# B&R Automation Studio project mappFramework (part 10)

#### Set_SetupTeardown.c - not listed in the package file held
```c
#include <bur/plctypes.h>

#ifdef _DEFAULT_INCLUDES
#include <AsDefault.h>
#endif

#include "UnitTest.h"
#include <stdbool.h>
#include <string.h>

_SETUP_SET(void)
{
	/* TODO:  add code running before test set here */
	TEST_DONE;
}

_TEARDOWN_SET(void)
{
	/* TODO:  add code running after test set here */
	TEST_DONE;
}

_SETUP_TEST(void)
{
    TestState = 0;
    FileNumber = 0;

    HmiFile_UT.Parameters.Fifo.Enable = false;
    HmiFile_UT.Parameters.Fifo.ScanInterval = 60;
    strcpy(HmiFile_UT.Parameters.Fifo.DeviceName, "mappUserXFiles");

    switch (SetupState)
    {
        case 0:
            DirInfo_UT.enable = true;
            DirInfo_UT.pDevice = (UDINT)&"mappUserXFiles";
            DirInfo_UT.pPath = (UDINT)&"";
            DirInfo(&DirInfo_UT);
            TEST_BUSY_CONDITION(DirInfo_UT.status == 65535);
            TEST_ABORT_CONDITION(DirInfo_UT.status != 0);
            NumberOfFiles = DirInfo_UT.filenum;
            CurrentFile = 0;
            SetupState = (NumberOfFiles == 0) ? 100 : 1;
            break;

        case 1:
            DirRead_UT.enable = true;
            DirRead_UT.pDevice = DirInfo_UT.pDevice;
            DirRead_UT.entry = 0;
            DirRead_UT.option = fiFILE;
            DirRead_UT.pData = (UDINT)&fileInfo;
            DirRead_UT.data_len = sizeof(fileInfo);
            DirRead(&DirRead_UT);
            TEST_BUSY_CONDITION(DirRead_UT.status == 65535);
            TEST_ABORT_CONDITION(DirRead_UT.status != 0);
            SetupState = 2;
            break;

        case 2:
            FileDelete_UT.enable = true;
            FileDelete_UT.pDevice = DirInfo_UT.pDevice;
            FileDelete_UT.pName = (UDINT)&fileInfo.Filename;
            FileDelete(&FileDelete_UT);
            TEST_BUSY_CONDITION(FileDelete_UT.status == 65535);
            TEST_ABORT_CONDITION(FileDelete_UT.status != 0);

            CurrentFile++;
            SetupState = (CurrentFile >= NumberOfFiles) ? 100 : 1;
            break;

        case 100:
            TEST_DONE;
    }
    TEST_BUSY;
}

_TEARDOWN_TEST(void)
{
    HmiFile_UT.Parameters.Fifo.Enable = false;
    HmiFile_UT.Parameters.Fifo.ScanInterval = 60;
    TestState = 0;
    SetupState = 0;
	TEST_DONE;
}

_TEST FIFO_20(void)
{
    switch (TestState)
    {
        // Arrange
        case 0:
            FileCreate_UT.enable = true;
            FileCreate_UT.pDevice = (UDINT)&"mappUserXFiles";
            snprintf2(FileName, sizeof(FileName), "TestFile%d.txt", FileNumber);
            FileCreate_UT.pFile = (UDINT)&FileName;
            FileCreate(&FileCreate_UT);

            TEST_BUSY_CONDITION(FileCreate_UT.status == 65535);
            TEST_ABORT_CONDITION(FileCreate_UT.status != 0);
            TestState = 1;
            break;

        case 1:
            FileClose_UT.enable = true;
            FileClose_UT.ident = FileCreate_UT.ident;
            FileClose(&FileClose_UT);

            TEST_BUSY_CONDITION(FileClose_UT.status == 65535);
            TEST_ABORT_CONDITION(FileClose_UT.status != 0);

            FileNumber++;
            TestState = (FileNumber >= 20) ? 10 : 0;
            break;

        // Act
        case 10:
            HmiFile_UT.Parameters.Fifo.Enable = true;
            strcpy(HmiFile_UT.Parameters.Fifo.DeviceName, "mappUserXFiles");
            HmiFile_UT.Parameters.Fifo.FifoType = FILE_FIFO_NUM_OF_FILES;
            HmiFile_UT.Parameters.Fifo.MaxNumberOfFiles = 10;
            HmiFile_UT.Parameters.Fifo.ScanInterval = 0;
            TEST_BUSY_CONDITION(HmiFile_UT.Status.DeleteStep == FILE_DELETE_WAIT);
            TestState = 100;
            break;

        // Assert
        case 100:
            TEST_BUSY_CONDITION(HmiFile_UT.Status.DeleteStep != FILE_DELETE_WAIT);
            HmiFile_UT.Parameters.Fifo.Enable = false;

            DirInfo_UT.enable = true;
            DirInfo_UT.pDevice = (UDINT)&"mappUserXFiles";
            DirInfo_UT.pPath = (UDINT)&"";
            DirInfo(&DirInfo_UT);
            TEST_BUSY_CONDITION(DirInfo_UT.status == 65535);
            TEST_ABORT_CONDITION(DirInfo_UT.status != 0);
            TEST_ASSERT_EQUAL_INT(HmiFile_UT.Parameters.Fifo.MaxNumberOfFiles, DirInfo_UT.filenum);
            TEST_DONE;
            break;
    }
    TEST_BUSY;
}

_TEST FIFO_60(void)
{
    switch (TestState)
    {
        // Arrange
        case 0:
            FileCreate_UT.enable = true;
            FileCreate_UT.pDevice = (UDINT)&"mappUserXFiles";
            snprintf2(FileName, sizeof(FileName), "TestFile%d.txt", FileNumber);
            FileCreate_UT.pFile = (UDINT)&FileName;
            FileCreate(&FileCreate_UT);

            TEST_BUSY_CONDITION(FileCreate_UT.status == 65535);
            TEST_ABORT_CONDITION(FileCreate_UT.status != 0);
            TestState = 1;
            break;

        case 1:
            FileClose_UT.enable = true;
            FileClose_UT.ident = FileCreate_UT.ident;
            FileClose(&FileClose_UT);

            TEST_BUSY_CONDITION(FileClose_UT.status == 65535);
            TEST_ABORT_CONDITION(FileClose_UT.status != 0);

            FileNumber++;
            TestState = (FileNumber >= 60) ? 10 : 0;
            break;

        // Act
        case 10:
            HmiFile_UT.Parameters.Fifo.Enable = true;
            strcpy(HmiFile_UT.Parameters.Fifo.DeviceName, "mappUserXFiles");
            HmiFile_UT.Parameters.Fifo.FifoType = FILE_FIFO_NUM_OF_FILES;
            HmiFile_UT.Parameters.Fifo.MaxNumberOfFiles = 15;
            HmiFile_UT.Parameters.Fifo.ScanInterval = 0;
            TEST_BUSY_CONDITION(HmiFile_UT.Status.DeleteStep == FILE_DELETE_WAIT);
            TestState = 100;
            break;

        // Assert
        case 100:
            TEST_BUSY_CONDITION(HmiFile_UT.Status.DeleteStep != FILE_DELETE_WAIT);
            HmiFile_UT.Parameters.Fifo.Enable = false;

            DirInfo_UT.enable = true;
            DirInfo_UT.pDevice = (UDINT)&"mappUserXFiles";
            DirInfo_UT.pPath = (UDINT)&"";
            DirInfo(&DirInfo_UT);
            TEST_BUSY_CONDITION(DirInfo_UT.status == 65535);
            TEST_ABORT_CONDITION(DirInfo_UT.status != 0);
            TEST_ASSERT_EQUAL_INT(HmiFile_UT.Parameters.Fifo.MaxNumberOfFiles, DirInfo_UT.filenum);
            TEST_DONE;
            break;

    }
    TEST_BUSY;
}

_TEST FIFO_140(void)
{
    switch (TestState)
    {
        // Arrange
        case 0:
            FileCreate_UT.enable = true;
            FileCreate_UT.pDevice = (UDINT)&"mappUserXFiles";
            snprintf2(FileName, sizeof(FileName), "TestFile%d.txt", FileNumber);
            FileCreate_UT.pFile = (UDINT)&FileName;
            FileCreate(&FileCreate_UT);

            TEST_BUSY_CONDITION(FileCreate_UT.status == 65535);
            TEST_ABORT_CONDITION(FileCreate_UT.status != 0);
            TestState = 1;
            break;

        case 1:
            FileClose_UT.enable = true;
            FileClose_UT.ident = FileCreate_UT.ident;
            FileClose(&FileClose_UT);

            TEST_BUSY_CONDITION(FileClose_UT.status == 65535);
            TEST_ABORT_CONDITION(FileClose_UT.status != 0);

            FileNumber++;
            TestState = (FileNumber >= 140) ? 10 : 0;
            break;

        // Act
        case 10:
            HmiFile_UT.Parameters.Fifo.Enable = true;
            strcpy(HmiFile_UT.Parameters.Fifo.DeviceName, "mappUserXFiles");
            HmiFile_UT.Parameters.Fifo.FifoType = FILE_FIFO_NUM_OF_FILES;
            HmiFile_UT.Parameters.Fifo.MaxNumberOfFiles = 15;
            HmiFile_UT.Parameters.Fifo.ScanInterval = 0;
            TEST_BUSY_CONDITION(HmiFile_UT.Status.DeleteStep == FILE_DELETE_WAIT);
            TestState = 100;
            break;

        // Assert
        case 100:
            TEST_BUSY_CONDITION(HmiFile_UT.Status.DeleteStep != FILE_DELETE_WAIT);
            HmiFile_UT.Parameters.Fifo.Enable = false;

            DirInfo_UT.enable = true;
            DirInfo_UT.pDevice = (UDINT)&"mappUserXFiles";
            DirInfo_UT.pPath = (UDINT)&"";
            DirInfo(&DirInfo_UT);
            TEST_BUSY_CONDITION(DirInfo_UT.status == 65535);
            TEST_ABORT_CONDITION(DirInfo_UT.status != 0);
            TEST_ASSERT_EQUAL_INT(HmiFile_UT.Parameters.Fifo.MaxNumberOfFiles, DirInfo_UT.filenum);
            TEST_DONE;
            break;

    }
    TEST_BUSY;
}

_TEST FIFO_MaxFiles60(void)
{
    switch (TestState)
    {
        // Arrange
        case 0:
            FileCreate_UT.enable = true;
            FileCreate_UT.pDevice = (UDINT)&"mappUserXFiles";
            snprintf2(FileName, sizeof(FileName), "TestFile%d.txt", FileNumber);
            FileCreate_UT.pFile = (UDINT)&FileName;
            FileCreate(&FileCreate_UT);

            TEST_BUSY_CONDITION(FileCreate_UT.status == 65535);
            TEST_ABORT_CONDITION(FileCreate_UT.status != 0);
            TestState = 1;
            break;

        case 1:
            FileClose_UT.enable = true;
            FileClose_UT.ident = FileCreate_UT.ident;
            FileClose(&FileClose_UT);

            TEST_BUSY_CONDITION(FileClose_UT.status == 65535);
            TEST_ABORT_CONDITION(FileClose_UT.status != 0);

            FileNumber++;
            TestState = (FileNumber >= 100) ? 10 : 0;
            break;

        // Act
        case 10:
            HmiFile_UT.Parameters.Fifo.Enable = true;
            strcpy(HmiFile_UT.Parameters.Fifo.DeviceName, "mappUserXFiles");
            HmiFile_UT.Parameters.Fifo.FifoType = FILE_FIFO_NUM_OF_FILES;
            HmiFile_UT.Parameters.Fifo.MaxNumberOfFiles = 60;
            HmiFile_UT.Parameters.Fifo.ScanInterval = 0;
            TEST_BUSY_CONDITION(HmiFile_UT.Status.DeleteStep == FILE_DELETE_WAIT);
            TestState = 100;
            break;

        // Assert
        case 100:
            TEST_BUSY_CONDITION(HmiFile_UT.Status.DeleteStep != FILE_DELETE_WAIT);
            HmiFile_UT.Parameters.Fifo.Enable = false;

            DirInfo_UT.enable = true;
            DirInfo_UT.pDevice = (UDINT)&"mappUserXFiles";
            DirInfo_UT.pPath = (UDINT)&"";
            DirInfo(&DirInfo_UT);
            TEST_BUSY_CONDITION(DirInfo_UT.status == 65535);
            TEST_ABORT_CONDITION(DirInfo_UT.status != 0);
            TEST_ASSERT_EQUAL_INT(HmiFile_UT.Parameters.Fifo.MaxNumberOfFiles, DirInfo_UT.filenum);
            TEST_DONE;
            break;

    }
    TEST_BUSY;
}

_TEST FIFO_MaxFiles120(void)
{
    switch (TestState)
    {
        // Arrange
        case 0:
            FileCreate_UT.enable = true;
            FileCreate_UT.pDevice = (UDINT)&"mappUserXFiles";
            snprintf2(FileName, sizeof(FileName), "TestFile%d.txt", FileNumber);
            FileCreate_UT.pFile = (UDINT)&FileName;
            FileCreate(&FileCreate_UT);

            TEST_BUSY_CONDITION(FileCreate_UT.status == 65535);
            TEST_ABORT_CONDITION(FileCreate_UT.status != 0);
            TestState = 1;
            break;

        case 1:
            FileClose_UT.enable = true;
            FileClose_UT.ident = FileCreate_UT.ident;
            FileClose(&FileClose_UT);

            TEST_BUSY_CONDITION(FileClose_UT.status == 65535);
            TEST_ABORT_CONDITION(FileClose_UT.status != 0);

            FileNumber++;
            TestState = (FileNumber >= 200) ? 10 : 0;
            break;

        // Act
        case 10:
            HmiFile_UT.Parameters.Fifo.Enable = true;
            strcpy(HmiFile_UT.Parameters.Fifo.DeviceName, "mappUserXFiles");
            HmiFile_UT.Parameters.Fifo.FifoType = FILE_FIFO_NUM_OF_FILES;
            HmiFile_UT.Parameters.Fifo.MaxNumberOfFiles = 120;
            HmiFile_UT.Parameters.Fifo.ScanInterval = 0;
            TEST_BUSY_CONDITION(HmiFile_UT.Status.DeleteStep == FILE_DELETE_WAIT);
            TestState = 100;
            break;

        // Assert
        case 100:
            TEST_BUSY_CONDITION(HmiFile_UT.Status.DeleteStep != FILE_DELETE_WAIT);
            HmiFile_UT.Parameters.Fifo.Enable = false;

            DirInfo_UT.enable = true;
            DirInfo_UT.pDevice = (UDINT)&"mappUserXFiles";
            DirInfo_UT.pPath = (UDINT)&"";
            DirInfo(&DirInfo_UT);
            TEST_BUSY_CONDITION(DirInfo_UT.status == 65535);
            TEST_ABORT_CONDITION(DirInfo_UT.status != 0);
            TEST_ASSERT_EQUAL_INT(HmiFile_UT.Parameters.Fifo.MaxNumberOfFiles, DirInfo_UT.filenum);
            TEST_DONE;
            break;

    }
    TEST_BUSY;
}

_TEST FIFO_MaxFolderSize_60Files(void)
{
    switch (TestState)
    {
        // Arrange
        case 0:
            FileCreate_UT.enable = true;
            FileCreate_UT.pDevice = (UDINT)&"mappUserXFiles";
            snprintf2(FileName, sizeof(FileName), "TestFile%d.txt", FileNumber);
            FileCreate_UT.pFile = (UDINT)&FileName;
            FileCreate(&FileCreate_UT);

            TEST_BUSY_CONDITION(FileCreate_UT.status == 65535);
            TEST_ABORT_CONDITION(FileCreate_UT.status != 0);
            TestState = 1;
            break;

        case 1:
            FileWrite_UT.enable = true;
            FileWrite_UT.ident = FileCreate_UT.ident;
            FileWrite_UT.offset = 0;
            FileWrite_UT.pSrc = &testData;
            FileWrite_UT.len = sizeof(testData);
            FileWrite(&FileWrite_UT);
            TEST_BUSY_CONDITION(FileWrite_UT.status == 65535);
            TEST_ABORT_CONDITION(FileWrite_UT.status != 0);
            TestState = 2;
            break;

        case 2:
            FileClose_UT.enable = true;
            FileClose_UT.ident = FileCreate_UT.ident;
            FileClose(&FileClose_UT);

            TEST_BUSY_CONDITION(FileClose_UT.status == 65535);
            TEST_ABORT_CONDITION(FileClose_UT.status != 0);

            FileNumber++;
            TestState = (FileNumber >= 60) ? 10 : 0;
            break;

        // Act
        case 10:
            HmiFile_UT.Parameters.Fifo.Enable = true;
            strcpy(HmiFile_UT.Parameters.Fifo.DeviceName, "mappUserXFiles");
            HmiFile_UT.Parameters.Fifo.FifoType = FILE_FIFO_SIZE_OF_FOLDER;
            HmiFile_UT.Parameters.Fifo.MaxFolderSize = 5 * 1024;
            HmiFile_UT.Parameters.Fifo.ScanInterval = 0;
            TEST_BUSY_CONDITION(HmiFile_UT.Status.DeleteStep == FILE_DELETE_WAIT);
            TestState = 100;
            break;

        // Assert
        case 100:
            TEST_BUSY_CONDITION(HmiFile_UT.Status.DeleteStep != FILE_DELETE_WAIT);
            HmiFile_UT.Parameters.Fifo.Enable = false;

            DirInfo_UT.enable = true;
            DirInfo_UT.pDevice = (UDINT)&"mappUserXFiles";
            DirInfo_UT.pPath = (UDINT)&"";
            DirInfo(&DirInfo_UT);
            TEST_BUSY_CONDITION(DirInfo_UT.status == 65535);
            TEST_ABORT_CONDITION(DirInfo_UT.status != 0);
            TEST_ASSERT_EQUAL_INT(5, DirInfo_UT.filenum);
            TEST_DONE;
            break;

    }
    TEST_BUSY;
}

/*
B+R UnitTest: This is generated code.
Do not edit! Do not move!
Description: UnitTest Testprogramm infrastructure (TestSet).
LastUpdated: 2022-04-25 15:09:32Z
By B+R UnitTest Helper Version: 2.0.1.59
*/
UNITTEST_FIXTURES(fixtures)
{
    new_TestFixture("FIFO_20", FIFO_20),
    new_TestFixture("FIFO_60", FIFO_60),
    new_TestFixture("FIFO_140", FIFO_140),
    new_TestFixture("FIFO_MaxFiles60", FIFO_MaxFiles60),
    new_TestFixture("FIFO_MaxFiles120", FIFO_MaxFiles120),
    new_TestFixture("FIFO_MaxFolderSize_60Files", FIFO_MaxFolderSize_60Files),

};

UNITTEST_CALLER_COMPLETE_EXPLICIT(Set_SetupTeardown, "Set_SetupTeardown", setupTest, teardownTest, fixtures, setupSet, teardownSet, 0);
```

### Package Logical/UnitTest/Recipe - Package for mapp Recipe Framework

### Program Logical/UnitTest/Recipe/RecipeMgrUnitTest (ANSIC) - Unit Tests for FileMgr

- RecipeMgr.typ (reference to Logical/Infrastructure/Recipe/RecipeMgr/RecipeMgr.typ)

- RecipeMgr.var (reference to Logical/Infrastructure/Recipe/RecipeMgr/RecipeMgr.var)

- CommonVariables.var (reference to Logical/UnitTest/Common/CommonUT/CommonVariables.var)

- Set_Common.c (reference to Logical/UnitTest/Common/CommonUT/Set_Common.c)

#### variables.var - Name the suite and add PVs for the program
```iecst
(********************************************************************
 * COPYRIGHT --
 ********************************************************************
 * Program: utTemplate_automated
 * File: variables.var
 * Author: -
 * Created: -
 ********************************************************************
 * Local variables of program utTemplate_automated
 ********************************************************************)
(*Describe the test*)
VAR
	Testsuite : UtMgrTestSuite := (Name:='RecipeMgr',Description:='RecipeMgr Unit Tests',MetaInformation:='Meta');
END_VAR
(*Variables used in the tests*)
VAR
	cycleCount : {REDUND_UNREPLICABLE} USINT;
	pMachineSettings : REFERENCE TO MachineSettingsType;
	MachineSettingsSize : {REDUND_UNREPLICABLE} UDINT;
	pParameters : REFERENCE TO ParametersType;
	ParameterSize : {REDUND_UNREPLICABLE} UDINT;
	LastSelectedIndex : UDINT;
	SetupState : USINT;
	FileName : STRING[24];
	NumberOfFiles : UINT;
	CurrentFile : UINT;
	fileInfo : fiDIR_READ_DATA;
	DirInfo_UT : DirInfo;
	DirRead_UT : DirRead;
	FileDelete_UT : FileDelete;
	FileCopy_UT : FileCopy;
END_VAR
```

#### testSuite.h
```c
#ifndef __TEST_SUITE_H__
#define __TEST_SUITE_H__

bool RecipeExists(char* recipeName);
bool SelectRecipe(char* wantedRecipe);
testStatusEnum RemoveNonDefaultFiles(char* filter, char* selectFile, const USINT categoryIndex, const char* category);

#endif
```

#### testSuite.c
```c
/********************************************************************
 * COPYRIGHT --
 ********************************************************************
 * Program: -
 * Author:
 * Created:
 ********************************************************************
 * Test registration and handshake
 ********************************************************************/

#include <bur/plctypes.h>

#ifdef _DEFAULT_INCLUDES
#include <AsDefault.h>
#endif

#include "UnitTest.h"
#include <string.h>
#include <stdbool.h>

void _INIT initTestSuite(void)
{
	Testsuite.Enable = 1;
	utInit(&Testsuite);

	CommonTestsuite.Enable = 1;
	utInit(&CommonTestsuite);

	strcpy((char*)&FileDeviceName, "mappRecipeFiles");
	strcpy((char*)&TextNameSpace, "mappFramework/Recipe/Alarms");
	strcpy((char*)&TextID, "SaveFailed");
	strcpy((char*)&HmiRecipe.Parameters.DeviceName, "mappRecipeFiles");

	PV_xgetadr("RecipeMgr:MachineSettings", (void*)&pMachineSettings, &MachineSettingsSize);
	PV_xgetadr("RecipeMgr:Parameters", (void*)&pParameters, &ParameterSize);

	LastSelectedIndex++;
}

void _CYCLIC cyclicWithTest(void)
{
	utCyclic(&Testsuite);
	if (Testsuite.Informational.LastKnownPassedLocation.TestCaseName != 0)
		strcpy((char*)&LastTestCase, (char*)Testsuite.Informational.LastKnownPassedLocation.TestCaseName);
	if (Testsuite.Informational.LastKnownPassedLocation.TestSetName != 0)
		strcpy((char*)&LastTestSet, (char*)Testsuite.Informational.LastKnownPassedLocation.TestSetName);
	if (Testsuite.Informational.LastKnownPassedLocation.File != 0)
		strcpy((char*)&LastTestFile, (char*)Testsuite.Informational.LastKnownPassedLocation.File);
}

void _EXIT exitTestSuite(void)
{
	utExit(&Testsuite);
}

bool RecipeExists(char* recipeName)
{
	for (USINT i = 0; i<(sizeof(MpRecipeUIConnect.Recipe.List.Names)/sizeof(MpRecipeUIConnect.Recipe.List.Names[0])); i++)
	{
		if (strcmp(recipeName, MpRecipeUIConnect.Recipe.List.Names[i]) == 0)
		{
			return true;
		}
	}
	return false;
}

bool SelectRecipe(char* wantedRecipe)
{
	if (((MpRecipeUIConnect.Status != mpRECIPE_UI_STATUS_IDLE) && (MpRecipeUIConnect.Status != mpRECIPE_UI_STATUS_ERROR)) &&
		(strcmp(wantedRecipe, HmiRecipe.Status.SelectedRecipe) != 0)) return false;

	for (USINT i=0; i <= MpRecipeUIConnect.Recipe.List.MaxSelection; i++)
	{
		if (strcmp(wantedRecipe, MpRecipeUIConnect.Recipe.List.Names[i]) == 0)
			MpRecipeUIConnect.Recipe.List.SelectedIndex = i;
	}

	return (strcmp(wantedRecipe, HmiRecipe.Status.SelectedRecipe) == 0);
}

testStatusEnum RemoveNonDefaultFiles(char* filter, char* selectFile, const char* category)
{
	switch (SetupState)
	{
		case 0:
			DirInfo_UT.enable = true;
			DirInfo_UT.pDevice = (UDINT)&"mappRecipeFiles";
			DirInfo_UT.pPath = (UDINT)&"";
			DirInfo(&DirInfo_UT);
			TEST_BUSY_CONDITION(DirInfo_UT.status == 65535);
			TEST_ABORT_CONDITION(DirInfo_UT.status != 0);
			NumberOfFiles = DirInfo_UT.filenum;
			CurrentFile = 0;
			SetupState = (NumberOfFiles == 0) ? 100 : 1;
			break;

		case 1:
			DirRead_UT.enable = true;
			DirRead_UT.pDevice = DirInfo_UT.pDevice;
			DirRead_UT.entry = CurrentFile;
			DirRead_UT.option = fiFILE;
			DirRead_UT.pData = (UDINT)&fileInfo;
			DirRead_UT.data_len = sizeof(fileInfo);
			DirRead(&DirRead_UT);
			TEST_BUSY_CONDITION(DirRead_UT.status == 65535);
			TEST_ABORT_CONDITION(DirRead_UT.status != 0);
			SetupState = 2;
			break;

		case 2:
			if ((strcmp("Default.par", (char*)fileInfo.Filename) == 0) ||
				(strcmp("Machine.mcfg", (char*)fileInfo.Filename) == 0))
			{
				CurrentFile++;
				SetupState = (CurrentFile >= NumberOfFiles) ? 10 : 1;
				break;
			}
			FileDelete_UT.enable = true;
			FileDelete_UT.pDevice = DirInfo_UT.pDevice;
			FileDelete_UT.pName = (UDINT)&fileInfo.Filename;
			FileDelete(&FileDelete_UT);
			TEST_BUSY_CONDITION(FileDelete_UT.status == 65535);
			TEST_ABORT_CONDITION(FileDelete_UT.status != 0);

			NumberOfFiles--;
			SetupState = (CurrentFile >= NumberOfFiles) ? 10 : 1;
			break;

		case 10:
			strcpy((char*)&HmiRecipe.Parameters.DeviceName, "mappRecipeFiles");
			strcpy((char*)&MpRecipeUIConnect.Recipe.Filter, filter);
			MpRecipeUIConnect.Recipe.Refresh = true;
			strcpy((char*)&HmiRecipe.Parameters.Category, category);
			TEST_BUSY_CONDITION(MpRecipeUIConnect.Status != mpRECIPE_UI_STATUS_REFRESH)
			MpRecipeUIConnect.Recipe.Refresh = false;
			SetupState = 11;
			break;

		case 11:
			TEST_BUSY_CONDITION(MpRecipeUIConnect.Status != mpRECIPE_UI_STATUS_IDLE)
			TEST_BUSY_CONDITION(!RecipeExists(selectFile));
			TEST_BUSY_CONDITION(HmiRecipe.Status.HMIcommand != REC_HMI_WAIT)
			TEST_ABORT_CONDITION(pParameters == NULL);
			SetupState = 100;
			break;

		case 100:
			cycleCount = 0;
			TestState = TEST_ARRANGE;
			SetupState = 0;
			TEST_DONE;
	}
	TEST_BUSY;
}
```

#### autoGeneratedFile.c - Auto generated code - list of all test sets in the program
```c
/*
B+R UnitTest: This is generated code.
Do not edit! Do not move!
Description: UnitTest Testprogramm infrastructure (List of TestSets).
LastUpdated: 2022-11-02 11:34:44Z
By B+R UnitTest Helper Version: 2.0.1.59
*/
#include "UnitTest.h"

UNITTEST_TESTSET_DECLARATION  Set_Common;
UNITTEST_TESTSET_DECLARATION  Set_RecipeParameters;
UNITTEST_TESTSET_DECLARATION  Set_RecipeMachineSettings;

UNITTEST_TESTSET_FIXTURES(utTestSets)
{
	new_TestSet(Set_Common),
	new_TestSet(Set_RecipeParameters),
	new_TestSet(Set_RecipeMachineSettings),
};
UNTITTEST_TESTSET_HANDLER();
```

#### Set_RecipeParameters.c
```c
#include <bur/plctypes.h>

#ifdef _DEFAULT_INCLUDES
#include <AsDefault.h>
#endif

#include "UnitTest.h"
#include <stdbool.h>
#include <string.h>
#include <stdlib.h>
#include "testSuite.h"

#define TIMEOUT_TEST_CASE                                   \
    if (cycleCount >= 254)                                  \
    {                                                       \
        char abortMessage[80];                              \
        char substate[10];                                  \
        memset(abortMessage, 0, sizeof(abortMessage));      \
        memset(substate, 0, sizeof(substate));              \
        itoa(ActSubState, substate, 10);                    \
        strcpy(abortMessage, "Timeout in ActSubState = ");  \
        strcat(abortMessage, substate);                     \
        TEST_FAIL(abortMessage);                            \
        TEST_DONE;                                          \
    }

_SETUP_SET(void)
{
    return RemoveNonDefaultFiles("*.par", "Default.par", PARAMETERS_CATEGORY);
}

_TEARDOWN_SET(void)
{
    SetupState = 0;
    TEST_DONE;
}

_SETUP_TEST(void)
{
    ArrangeSubState = 0;
    ActSubState = 0;
    AssertSubState = 0;
    return RemoveNonDefaultFiles("*.par", "Default.par", PARAMETERS_CATEGORY);
}

_TEARDOWN_TEST(void)
{
    memset(&HmiRecipe.Commands, 0, sizeof(HmiRecipe.Commands));
    MpRecipeUIConnect.Recipe.Load = false;
    TEST_BUSY_CONDITION(!SelectRecipe("Default.par"));

    if (MpRecipeUIConnect.Status == mpRECIPE_UI_STATUS_ERROR)
    {
        MpRecipeUIConnect.Recipe.Refresh = true;
    }
    TEST_BUSY_CONDITION(MpRecipeUIConnect.Status != mpRECIPE_UI_STATUS_IDLE)
    MpRecipeUIConnect.Recipe.Refresh = false;

    TEST_DONE;
}

_CYCLIC_SET(void)
{
    cycleCount++;
}

_TEST DefaultValues(void)
{
    TIMEOUT_TEST_CASE
    switch (TestState)
    {
        case TEST_ARRANGE:
            // set MachineSettings through the pointer
            memset(pParameters, 0, sizeof(*pParameters));
            TEST_BUSY_CONDITION(!SelectRecipe("Default.par"));
            TEST_BUSY_CONDITION(MpRecipeUIConnect.Status != mpRECIPE_UI_STATUS_IDLE);
            TEST_BUSY_CONDITION(HmiRecipe.Status.HMIcommand != REC_HMI_WAIT);
            TestState = TEST_ACT;
            break;

        case TEST_ACT:
            switch (ActSubState)
            {
                case 0:
                    MpRecipeUIConnect.Recipe.Load = true;
                    TEST_BUSY_CONDITION(MpRecipeUIConnect.Status != mpRECIPE_UI_STATUS_LOAD);
                    MpRecipeUIConnect.Recipe.Load = false;
                    ActSubState = 1;
                    break;

                case 1:
                    TEST_BUSY_CONDITION(MpRecipeUIConnect.Status != mpRECIPE_UI_STATUS_IDLE);
                    HmiRecipe.Commands.LoadRecipe = true;
                    TEST_BUSY_CONDITION(HmiRecipe.Status.ProductRecipeLoaded == true);
                    TEST_BUSY_CONDITION(HmiRecipe.Status.HMIcommand == REC_HMI_WAIT);
                    HmiRecipe.Commands.LoadRecipe = false;
                    ActSubState = 2;
                    break;

                case 2:
                    TEST_BUSY_CONDITION(HmiRecipe.Status.ProductRecipeLoaded == false);
                    TEST_BUSY_CONDITION(HmiRecipe.Status.HMIcommand != REC_HMI_WAIT);
                    TestState = TEST_ASSERT;
                    break;
            }
            break;

        case TEST_ASSERT:
            TEST_ASSERT(Parameters.AddParametersHere1);
            TEST_ASSERT_EQUAL_STRING("two", Parameters.AddParametersHere2);
            TEST_ASSERT_DOUBLE_WITHIN(0.0001, 3.3, Parameters.AddParametersHere3);
            TEST_ASSERT_DOUBLE_WITHIN(0.0001, 4.4, Parameters.AddParametersHere4);
            TEST_ASSERT_DOUBLE_WITHIN(0.0001, 5.5, Parameters.AddParametersHere5);
            TEST_DONE;
            break;
    }
    TEST_BUSY;
}

_TEST CreateNew(void)
{
    TIMEOUT_TEST_CASE
    switch (TestState)
    {
        case TEST_ARRANGE:
            strcpy(HmiRecipe.Parameters.FileName, "test");
            TEST_BUSY_CONDITION(MpRecipeUIConnect.Status != mpRECIPE_UI_STATUS_IDLE);
            TEST_BUSY_CONDITION(HmiRecipe.Status.HMIcommand != REC_HMI_WAIT);
            TestState = TEST_ACT;
            break;

        case TEST_ACT:
            if (MpRecipeUIConnect.Status == mpRECIPE_UI_STATUS_ERROR)
            {
                TEST_FAIL("MpRecipeUIConnect in error state");
            }
            switch (ActSubState)
            {
                case 0:
                    HmiRecipe.Commands.CreateRecipe = true;
                    TEST_BUSY_CONDITION(MpRecipeUIConnect.Status != mpRECIPE_UI_STATUS_CREATE);
                    HmiRecipe.Commands.CreateRecipe = false;
                    ActSubState = 1;
                    break;

                case 1:
                    TEST_BUSY_CONDITION(MpRecipeUIConnect.Status != mpRECIPE_UI_STATUS_IDLE);
                    TEST_BUSY_CONDITION(HmiRecipe.Status.ProductRecipeLoaded == false);
                    ActSubState = 2;
                    break;

                case 2:
                    TEST_BUSY_CONDITION(MpRecipeUIConnect.Status == mpRECIPE_UI_STATUS_REFRESH);
                    ActSubState = 3;
                    break;

                case 3:
                    TEST_BUSY_CONDITION(MpRecipeUIConnect.Status != mpRECIPE_UI_STATUS_IDLE);
                    TestState = TEST_ASSERT;
                    break;
            }
            break;

        case TEST_ASSERT:
            TEST_ASSERT(RecipeExists("test.par"));
            TEST_DONE;
            break;
    }

    TEST_BUSY;
}

_TEST CreateExisting(void)
{
    TIMEOUT_TEST_CASE
    switch (TestState)
    {
        case TEST_ARRANGE:
            strcpy(HmiRecipe.Parameters.FileName, "Default");
            TEST_BUSY_CONDITION(MpRecipeUIConnect.Status != mpRECIPE_UI_STATUS_IDLE);
            TEST_BUSY_CONDITION(HmiRecipe.Status.HMIcommand != REC_HMI_WAIT);
            TestState = TEST_ACT;
            break;

        case TEST_ACT:
            TestState = TEST_ASSERT;
            break;

        case TEST_ASSERT:
            HmiRecipe.Commands.CreateRecipe = false;
            TEST_ASSERT(HmiRecipe.Status.FileDuplicate);
            TEST_ASSERT(RecipeExists("Default.par"));
            TEST_DONE;
            break;
    }

    TEST_BUSY;
}

_TEST CreateNonExisting(void)
{
    TIMEOUT_TEST_CASE

    switch (TestState)
    {
        case TEST_ARRANGE:
            strcpy(HmiRecipe.Parameters.FileName, "test2");
            TEST_BUSY_CONDITION(MpRecipeUIConnect.Status != mpRECIPE_UI_STATUS_IDLE);
            TEST_BUSY_CONDITION(HmiRecipe.Status.HMIcommand != REC_HMI_WAIT);
            TestState = TEST_ACT;
            break;

        case TEST_ACT:
            TestState = TEST_ASSERT;
            break;

        case TEST_ASSERT:
            HmiRecipe.Commands.CreateRecipe = false;
            TEST_ASSERT(!HmiRecipe.Status.FileDuplicate);
            TEST_ASSERT(!RecipeExists("test2.par"));
            TEST_DONE;
            break;
    }
    TEST_BUSY;
}

_TEST CreateActive(void)
{
    TIMEOUT_TEST_CASE
    switch (TestState)
    {
        case TEST_ARRANGE:
            strcpy(HmiRecipe.Parameters.FileName, strtok(HmiRecipe.Status.LastLoadedProductRecipe, "."));
            TEST_BUSY_CONDITION(MpRecipeUIConnect.Status != mpRECIPE_UI_STATUS_IDLE);
            TEST_BUSY_CONDITION(HmiRecipe.Status.HMIcommand != REC_HMI_WAIT);
            TestState = TEST_ACT;
            break;

        case TEST_ACT:
            TestState = TEST_ASSERT;
            break;

        case TEST_ASSERT:
            HmiRecipe.Commands.CreateRecipe = false;
            TEST_ASSERT(HmiRecipe.Status.FileDuplicate);
            TEST_ASSERT(RecipeExists(HmiRecipe.Status.LastLoadedProductRecipe));
            TEST_DONE;
            break;
    }
    TEST_BUSY;
}

_TEST PreviewShouldNotAffectActive(void)
{
    TIMEOUT_TEST_CASE
    switch (TestState)
    {
        case TEST_ARRANGE:
            ParametersEdit.AddParametersHere1 = false;
            strcpy(ParametersEdit.AddParametersHere2, "testing preview");
            ParametersEdit.AddParametersHere3 = 12.56;
            ParametersEdit.AddParametersHere4 = 134.876;
            ParametersEdit.AddParametersHere5 = 87.4567;
            strcpy(HmiRecipe.Parameters.FileName, "preview");
            TEST_BUSY_CONDITION(MpRecipeUIConnect.Status != mpRECIPE_UI_STATUS_IDLE);
            TEST_BUSY_CONDITION(HmiRecipe.Status.HMIcommand != REC_HMI_WAIT);
            TestState = TEST_ACT;
            break;

        case TEST_ACT:
            if (MpRecipeUIConnect.Status == mpRECIPE_UI_STATUS_ERROR)
            {
                TEST_FAIL("MpRecipeUIConnect in error state");
                TEST_DONE;
            }
            switch (ActSubState)
            {
                case 0:
                    HmiRecipe.Commands.CreateRecipe = true;
                    TEST_BUSY_CONDITION(MpRecipeUIConnect.Status != mpRECIPE_UI_STATUS_CREATE);
                    HmiRecipe.Commands.CreateRecipe = false;
                    ActSubState = 1;
                    break;

                case 1:
                    TEST_BUSY_CONDITION(MpRecipeUIConnect.Status != mpRECIPE_UI_STATUS_IDLE);
                    TEST_BUSY_CONDITION(HmiRecipe.Status.ProductRecipeLoaded == false);
                    ActSubState = 2;
                    break;

                case 2:
                    TEST_BUSY_CONDITION(MpRecipeUIConnect.Status == mpRECIPE_UI_STATUS_REFRESH);
                    ActSubState = 3;
                    break;

                case 3:
                    TEST_BUSY_CONDITION(MpRecipeUIConnect.Status != mpRECIPE_UI_STATUS_IDLE);
                    TEST_BUSY_CONDITION(!SelectRecipe("preview.par"));
                    ActSubState = 4;
                    break;

                case 4:
                    TEST_BUSY_CONDITION(!SelectRecipe("preview.par"));
                    MpRecipeUIConnect.Recipe.Load = true;
                    TEST_BUSY_CONDITION(MpRecipeUIConnect.Status != mpRECIPE_UI_STATUS_LOAD);
                    MpRecipeUIConnect.Recipe.Load = false;
                    ActSubState = 5;
                    break;

                case 5:
                    TEST_BUSY_CONDITION(MpRecipeUIConnect.Status != mpRECIPE_UI_STATUS_IDLE);
                    TestState = TEST_ASSERT;
                    break;
            }
            break;

        case TEST_ASSERT:
            // check if preview affects the active parameters
            TEST_ASSERT(Parameters.AddParametersHere1);
            TEST_ASSERT_EQUAL_STRING("two", Parameters.AddParametersHere2);
            TEST_ASSERT_DOUBLE_WITHIN(0.0001, 3.3, Parameters.AddParametersHere3);
            TEST_ASSERT_DOUBLE_WITHIN(0.0001, 4.4, Parameters.AddParametersHere4);
            TEST_ASSERT_DOUBLE_WITHIN(0.0001, 5.5, Parameters.AddParametersHere5);
            TEST_DONE;
            break;
    }
    TEST_BUSY;
}

_TEST Preview(void)
{
    TIMEOUT_TEST_CASE

    switch (TestState)
    {
        case TEST_ARRANGE:
            ParametersEdit.AddParametersHere1 = false;
            strcpy(ParametersEdit.AddParametersHere2, "testing preview");
            ParametersEdit.AddParametersHere3 = 12.56;
            ParametersEdit.AddParametersHere4 = 134.876;
            ParametersEdit.AddParametersHere5 = 87.4567;
            strcpy(HmiRecipe.Parameters.FileName, "preview");
            TEST_BUSY_CONDITION(MpRecipeUIConnect.Status != mpRECIPE_UI_STATUS_IDLE);
            TEST_BUSY_CONDITION(HmiRecipe.Status.HMIcommand != REC_HMI_WAIT);
            TestState = TEST_ACT;
            break;

        case TEST_ACT:
            if (MpRecipeUIConnect.Status == mpRECIPE_UI_STATUS_ERROR)
            {
                TEST_FAIL("MpRecipeUIConnect in error state");
                TEST_DONE;
            }
            switch (ActSubState)
            {
                case 0:
                    HmiRecipe.Commands.CreateRecipe = true;
                    TEST_BUSY_CONDITION(MpRecipeUIConnect.Status != mpRECIPE_UI_STATUS_CREATE);
                    HmiRecipe.Commands.CreateRecipe = false;
                    ActSubState = 1;
                    break;

                case 1:
                    TEST_BUSY_CONDITION(MpRecipeUIConnect.Status != mpRECIPE_UI_STATUS_IDLE);
                    TEST_BUSY_CONDITION(HmiRecipe.Status.ProductRecipeLoaded == false);
                    ActSubState = 2;
                    break;

                case 2:
                    TEST_BUSY_CONDITION(MpRecipeUIConnect.Status == mpRECIPE_UI_STATUS_REFRESH);
                    ActSubState = 3;
                    break;

                case 3:
                    TEST_BUSY_CONDITION(MpRecipeUIConnect.Status != mpRECIPE_UI_STATUS_IDLE);
                    TEST_BUSY_CONDITION(!SelectRecipe("preview.par"));
                    ActSubState = 4;
                    break;

                case 4:
                    TEST_BUSY_CONDITION(!SelectRecipe("preview.par"));
                    MpRecipeUIConnect.Recipe.Load = true;
                    TEST_BUSY_CONDITION(MpRecipeUIConnect.Status != mpRECIPE_UI_STATUS_LOAD);
                    MpRecipeUIConnect.Recipe.Load = false;
                    ActSubState = 5;
                    break;

                case 5:
                    TEST_BUSY_CONDITION(MpRecipeUIConnect.Status != mpRECIPE_UI_STATUS_IDLE);
                    TestState = TEST_ASSERT;
                    break;
            }
            break;

        case TEST_ASSERT:
            TEST_ASSERT(!ParametersPreview.AddParametersHere1);
            TEST_ASSERT_EQUAL_STRING("testing preview", ParametersPreview.AddParametersHere2);
            TEST_ASSERT_DOUBLE_WITHIN(0.0001, 12.56, ParametersPreview.AddParametersHere3);
            TEST_ASSERT_DOUBLE_WITHIN(0.0001, 134.876, ParametersPreview.AddParametersHere4);
            TEST_ASSERT_DOUBLE_WITHIN(0.0001, 87.4567, ParametersPreview.AddParametersHere5);

            TEST_DONE;
            break;
    }
    TEST_BUSY;
}

_TEST Delete(void)
{
    TIMEOUT_TEST_CASE
    switch (TestState)
    {
        case TEST_ARRANGE:
            switch (ArrangeSubState)
            {
                case 0:
                    strcpy(HmiRecipe.Parameters.FileName, "test");
                    TEST_BUSY_CONDITION(MpRecipeUIConnect.Status != mpRECIPE_UI_STATUS_IDLE);
                    TEST_BUSY_CONDITION(HmiRecipe.Status.HMIcommand != REC_HMI_WAIT);
                    ArrangeSubState = 1;
                    break;

                case 1:
                    HmiRecipe.Commands.CreateRecipe = true;
                    TEST_BUSY_CONDITION(MpRecipeUIConnect.Status != mpRECIPE_UI_STATUS_CREATE);
                    HmiRecipe.Commands.CreateRecipe = false;
                    ArrangeSubState = 2;
                    break;

                case 2:
                    TEST_BUSY_CONDITION(MpRecipeUIConnect.Status != mpRECIPE_UI_STATUS_IDLE);
                    TEST_BUSY_CONDITION(HmiRecipe.Status.ProductRecipeLoaded == false);
                    ArrangeSubState = 3;
                    break;

                case 3:
                    TEST_BUSY_CONDITION(MpRecipeUIConnect.Status == mpRECIPE_UI_STATUS_REFRESH);
                    ArrangeSubState = 4;
                    break;

                case 4:
                    TEST_BUSY_CONDITION(MpRecipeUIConnect.Status != mpRECIPE_UI_STATUS_IDLE);
                    ArrangeSubState = 5;
                    break;

                case 5:
                    TEST_BUSY_CONDITION(!SelectRecipe("test.par"));
                    TEST_BUSY_CONDITION(MpRecipeUIConnect.Status != mpRECIPE_UI_STATUS_IDLE);
                    TEST_BUSY_CONDITION(HmiRecipe.Status.HMIcommand != REC_HMI_WAIT);
                    TestState = TEST_ACT;
                    break;
            }
            break;

        case TEST_ACT:
            if (MpRecipeUIConnect.Status == mpRECIPE_UI_STATUS_ERROR)
            {
                TEST_FAIL("MpRecipeUIConnect in error state");
                TEST_DONE;
            }
            switch (ActSubState) {
                case 0:
                    MpRecipeUIConnect.Recipe.Delete = true;
                    TEST_BUSY_CONDITION(MpRecipeUIConnect.MessageBox.LayerStatus != 0);
                    MpRecipeUIConnect.Recipe.Delete = false;
                    MpRecipeUIConnect.MessageBox.Confirm = true;
                    ActSubState = 1;
                    break;

                case 1:
                    MpRecipeUIConnect.MessageBox.Confirm = false;
                    TEST_BUSY_CONDITION(MpRecipeUIConnect.MessageBox.LayerStatus == 0)
                    TEST_BUSY_CONDITION(MpRecipeUIConnect.Status == mpRECIPE_UI_STATUS_IDLE);
                    ActSubState = 2;
                    break;

                case 2:
                    TEST_BUSY_CONDITION(MpRecipeUIConnect.Status != mpRECIPE_UI_STATUS_IDLE);
                    ActSubState = 3;
                    break;

                case 3:
                    TEST_BUSY_CONDITION(MpRecipeUIConnect.Status == mpRECIPE_UI_STATUS_REFRESH);
                    ActSubState = 4;
                    break;

                case 4:
                    TEST_BUSY_CONDITION(MpRecipeUIConnect.Status != mpRECIPE_UI_STATUS_IDLE);
                    TestState = TEST_ASSERT;
                    break;
            }
            break;

        case TEST_ASSERT:
            TEST_ASSERT(!RecipeExists("test.par"));
            TEST_DONE;
            break;
    }
    TEST_BUSY;
}

_TEST Invalid(void)
{
    TIMEOUT_TEST_CASE
    switch (TestState)
    {
        case TEST_ARRANGE:
            switch (ArrangeSubState) {
                case 0:
                    FileCopy_UT.enable = true;
                    FileCopy_UT.pSrcDev = "mappRecipeFiles";
                    FileCopy_UT.pSrc = "CSVformat\\Default.par";
                    FileCopy_UT.pDestDev = "mappRecipeFiles";
                    FileCopy_UT.pDest = "Invalid.par";
                    FileCopy_UT.option= fiOVERWRITE;
                    FileCopy(&FileCopy_UT);
                    TEST_BUSY_CONDITION(FileCopy_UT.status == 65535);
                    FileCopy_UT.enable = false;
                    FileCopy(&FileCopy_UT);
                    ArrangeSubState = 1;
                    break;

                case 1:
                    MpRecipeUIConnect.Recipe.Refresh = true;
                    TEST_BUSY_CONDITION(MpRecipeUIConnect.Status == mpRECIPE_UI_STATUS_IDLE);
                    MpRecipeUIConnect.Recipe.Refresh = false;
                    ArrangeSubState = 2;
                    break;

                case 2:
                    TEST_BUSY_CONDITION(MpRecipeUIConnect.Status == mpRECIPE_UI_STATUS_REFRESH);
                    ArrangeSubState = 3;
                    break;

                case 3:
                    TEST_BUSY_CONDITION(!SelectRecipe("Invalid.par"));
                    TEST_BUSY_CONDITION(MpRecipeUIConnect.Status != mpRECIPE_UI_STATUS_IDLE);
                    TEST_BUSY_CONDITION(HmiRecipe.Status.HMIcommand != REC_HMI_WAIT);
                    TestState = TEST_ACT;
                    break;
            }
            break;

        case TEST_ACT:
            switch (ActSubState)
            {
                case 0:
                    MpRecipeUIConnect.Recipe.Load = true;
                    TEST_BUSY_CONDITION(MpRecipeUIConnect.Status != mpRECIPE_UI_STATUS_LOAD);
                    MpRecipeUIConnect.Recipe.Load = false;
                    ActSubState = 1;
                    break;

                case 1:
                    TEST_BUSY_CONDITION(MpRecipeUIConnect.Status == mpRECIPE_UI_STATUS_LOAD);
                    TestState = TEST_ASSERT;
                    break;
            }
            break;

        case TEST_ASSERT:
            TEST_ASSERT_EQUAL_INT(mpRECIPE_UI_STATUS_ERROR, MpRecipeUIConnect.Status);
            TEST_DONE;
            break;
    }
    TEST_BUSY;
}

SKIP_TEST EditActive(void)
{
    TIMEOUT_TEST_CASE
    switch (TestState)
    {
        case TEST_ARRANGE:
            TEST_BUSY_CONDITION(!SelectRecipe("Default.par"));
            LastSelectedIndex++;
            TEST_BUSY_CONDITION(HmiRecipe.Status.HMIcommand != REC_HMI_WAIT);
            TEST_BUSY_CONDITION(MpRecipeUIConnect.Status != mpRECIPE_UI_STATUS_IDLE);

            ParametersEdit.AddParametersHere1 = false;
            strcpy(ParametersEdit.AddParametersHere2, "testing editing active");
            ParametersEdit.AddParametersHere3 = 12.56;
            ParametersEdit.AddParametersHere4 = 134.876;
            ParametersEdit.AddParametersHere5 = 87.4567;
            strcpy(HmiRecipe.Parameters.FileName, "editActive");
            TestState = TEST_ACT;
            break;

        case TEST_ACT:
            if (MpRecipeUIConnect.Status == mpRECIPE_UI_STATUS_ERROR)
            {
                TEST_FAIL("MpRecipeUIConnect in error state");
                TEST_DONE;
            }
            switch (ActSubState)
            {
                case 0:
                    HmiRecipe.Commands.CreateRecipe = true;
                    TEST_BUSY_CONDITION(MpRecipeUIConnect.Status != mpRECIPE_UI_STATUS_CREATE);
                    HmiRecipe.Commands.CreateRecipe = false;
                    ActSubState = 1;
                    break;

                case 1:
                    TEST_BUSY_CONDITION(MpRecipeUIConnect.Status != mpRECIPE_UI_STATUS_IDLE);
                    TEST_BUSY_CONDITION(HmiRecipe.Status.ProductRecipeLoaded == false);
                    ActSubState = 2;
                    break;

                case 2:
                    TEST_BUSY_CONDITION(MpRecipeUIConnect.Status == mpRECIPE_UI_STATUS_REFRESH);
                    ActSubState = 3;
                    break;

                case 3:
                    TEST_BUSY_CONDITION(MpRecipeUIConnect.Status != mpRECIPE_UI_STATUS_IDLE);
                    TEST_BUSY_CONDITION(HmiRecipe.Status.ProductRecipeLoaded == false);
                    TEST_BUSY_CONDITION(!SelectRecipe("editActive.par"));
                    ActSubState = 4;
                    break;

                case 4:
                    MpRecipeUIConnect.Recipe.Load = true;
                    TEST_BUSY_CONDITION(MpRecipeUIConnect.Status != mpRECIPE_UI_STATUS_LOAD);
                    MpRecipeUIConnect.Recipe.Load = false;
                    ActSubState = 5;
                    break;

                case 5:
                    TEST_BUSY_CONDITION(MpRecipeUIConnect.Status != mpRECIPE_UI_STATUS_IDLE);
                    ParametersEdit.AddParametersHere1 = true;
                    strcpy(ParametersEdit.AddParametersHere2, "edited active");
                    ParametersEdit.AddParametersHere3 = 52.56;
                    ParametersEdit.AddParametersHere4 = 184.876;
                    ParametersEdit.AddParametersHere5 = 587.4567;
                    ActSubState = 6;
                    break;

                case 6:
                    HmiRecipe.Commands.SaveSelectedRecipe = true;
                    TEST_BUSY_CONDITION(HmiRecipe.Status.HMIcommand == REC_HMI_WAIT);
                    HmiRecipe.Commands.SaveSelectedRecipe = false;
                    ActSubState = 7;
                    break;

                case 7:
                    TEST_BUSY_CONDITION(HmiRecipe.Status.HMIcommand != REC_HMI_WAIT);
                    TEST_BUSY_CONDITION(MpRecipeUIConnect.Status != mpRECIPE_UI_STATUS_IDLE);
                    TestState = TEST_ASSERT;
                    break;
            }
            break;

        case TEST_ASSERT:
            TEST_ASSERT(Parameters.AddParametersHere1);
            TEST_ASSERT_EQUAL_STRING("edited active", Parameters.AddParametersHere2);
            TEST_ASSERT_DOUBLE_WITHIN(0.0001, 52.56, Parameters.AddParametersHere3);
            TEST_ASSERT_DOUBLE_WITHIN(0.0001, 184.876, Parameters.AddParametersHere4);
            TEST_ASSERT_DOUBLE_WITHIN(0.0001, 587.4567, Parameters.AddParametersHere5);

            TEST_DONE;
            break;
    }
    TEST_BUSY;
}

/*
B+R UnitTest: This is generated code.
Do not edit! Do not move!
Description: UnitTest Testprogramm infrastructure (TestSet).
LastUpdated: 2022-11-07 13:02:54Z
By B+R UnitTest Helper Version: 2.0.1.59
*/
UNITTEST_FIXTURES(fixtures)
{
    new_TestFixture("DefaultValues", DefaultValues),
    new_TestFixture("CreateNew", CreateNew),
    new_TestFixture("CreateExisting", CreateExisting),
    new_TestFixture("CreateNonExisting", CreateNonExisting),
    new_TestFixture("CreateActive", CreateActive),
    new_TestFixture("PreviewShouldNotAffectActive", PreviewShouldNotAffectActive),
    new_TestFixture("Preview", Preview),
    new_TestFixture("Delete", Delete),
    new_TestFixture("Invalid", Invalid),
    skipTestFixture("EditActive", EditActive),
};

UNITTEST_CALLER_COMPLETE_EXPLICIT(Set_RecipeParameters, "Set_RecipeParameters", setupTest, teardownTest, fixtures, setupSet, teardownSet, cyclicSetCaller);
```

#### Set_RecipeMachineSettings.c
```c
#include <bur/plctypes.h>

#ifdef _DEFAULT_INCLUDES
#include <AsDefault.h>
#endif

#include "UnitTest.h"
#include <stdbool.h>
#include <string.h>
#include <stdlib.h>
#include "testSuite.h"

#define TIMEOUT_TEST_CASE									\
	if (cycleCount >= 254)									\
	{														\
		char abortMessage[80];								\
		char substate[10];									\
		memset(abortMessage, 0, sizeof(abortMessage));		\
		memset(substate, 0, sizeof(substate));				\
		itoa(ActSubState, substate, 10);					\
		strcpy(abortMessage, "Timeout in ActSubState = ");	\
		strcat(abortMessage, substate);						\
		TEST_FAIL(abortMessage);							\
		TEST_DONE;											\
	}

_SETUP_SET(void)
{
	return RemoveNonDefaultFiles("*.mcfg", "Machine.mcfg", 1, MACHINE_CONFIGURATION_CATEGORY);
}

_TEARDOWN_SET(void)
{
	SetupState = 0;
	TEST_DONE;
}

_SETUP_TEST(void)
{
	ArrangeSubState = 0;
	ActSubState = 0;
	AssertSubState = 0;
	return RemoveNonDefaultFiles("*.mcfg", "Machine.mcfg", 1, MACHINE_CONFIGURATION_CATEGORY);
}

_TEARDOWN_TEST(void)
{
	memset(&HmiRecipe.Commands, 0, sizeof(HmiRecipe.Commands));
	MpRecipeUIConnect.Recipe.Load = false;
	TEST_BUSY_CONDITION(!SelectRecipe("Machine.mcfg"));

	if (MpRecipeUIConnect.Status == mpRECIPE_UI_STATUS_ERROR)
	{
		MpRecipeUIConnect.Recipe.Refresh = true;
	}
	TEST_BUSY_CONDITION(MpRecipeUIConnect.Status != mpRECIPE_UI_STATUS_IDLE)
	MpRecipeUIConnect.Recipe.Refresh = false;

	TEST_DONE;
}

_CYCLIC_SET(void)
{
	cycleCount++;
}

_TEST DefaultValues(void)
{
	TIMEOUT_TEST_CASE
	switch (TestState)
	{
		case TEST_ARRANGE:
			// set MachineSettings through the pointer
			memset(pMachineSettings, 0, sizeof(*pMachineSettings));
			TEST_BUSY_CONDITION(!SelectRecipe("Machine.mcfg"));
			TEST_BUSY_CONDITION(MpRecipeUIConnect.Status != mpRECIPE_UI_STATUS_IDLE);
			TEST_BUSY_CONDITION(HmiRecipe.Status.HMIcommand != REC_HMI_WAIT);
			TestState = TEST_ACT;
			break;

		case TEST_ACT:
			if (MpRecipeUIConnect.Status == mpRECIPE_UI_STATUS_ERROR)
			{
				TEST_FAIL("MpRecipeUIConnect in error state");
				TEST_DONE;
			}
			switch (ActSubState)
			{
				case 0:
					MpRecipeUIConnect.Recipe.Load = true;
					HmiRecipe.Commands.LoadRecipe = true;
					TEST_BUSY_CONDITION(HmiRecipe.Status.ConfigRecipeLoaded == true);
					TEST_BUSY_CONDITION(HmiRecipe.Status.HMIcommand == REC_HMI_WAIT);
					HmiRecipe.Commands.LoadRecipe = false;
					MpRecipeUIConnect.Recipe.Load = false;
					ActSubState = 1;
					break;
				case 1:
					TEST_BUSY_CONDITION(HmiRecipe.Status.ConfigRecipeLoaded == false);
					TEST_BUSY_CONDITION(HmiRecipe.Status.HMIcommand != REC_HMI_WAIT);
					TEST_BUSY_CONDITION(MpRecipeUIConnect.Status == mpRECIPE_UI_STATUS_LOAD);
					TestState = TEST_ASSERT;
					break;
			}
			break;

		case TEST_ASSERT:
			TEST_ASSERT_EQUAL_INT(11, MachineSettings.AddMachineSettingsHere1);
			TEST_ASSERT_EQUAL_INT(22, MachineSettings.AddMachineSettingsHere2);
			TEST_ASSERT_EQUAL_INT(true, MachineSettings.AddMachineSettingsHere3);
			TEST_ASSERT_DOUBLE_WITHIN(0.0001, 3.2999999, MachineSettings.AddMachineSettingsHere4);
			TEST_ASSERT_EQUAL_INT(44, MachineSettings.AddMachineSettingsHere5);
			TEST_DONE;
			break;
	}
	TEST_BUSY;

	TEST_DONE;
}
_TEST CreateNew(void)
{
	TIMEOUT_TEST_CASE
	switch (TestState)
	{
		case TEST_ARRANGE:
			strcpy(HmiRecipe.Parameters.FileName, "test");
			TEST_BUSY_CONDITION(MpRecipeUIConnect.Status != mpRECIPE_UI_STATUS_IDLE);
			TEST_BUSY_CONDITION(HmiRecipe.Status.HMIcommand != REC_HMI_WAIT);
			TestState = TEST_ACT;
			break;

		case TEST_ACT:
			if (MpRecipeUIConnect.Status == mpRECIPE_UI_STATUS_ERROR)
			{
				TEST_FAIL("MpRecipeUIConnect in error state");
				TEST_DONE;
			}
			switch (ActSubState)
			{
				case 0:
					HmiRecipe.Commands.CreateRecipe = true;
					TEST_BUSY_CONDITION(MpRecipeUIConnect.Status != mpRECIPE_UI_STATUS_CREATE);
					HmiRecipe.Commands.CreateRecipe = false;
					ActSubState = 1;
					break;

				case 1:
					TEST_BUSY_CONDITION(MpRecipeUIConnect.Status != mpRECIPE_UI_STATUS_IDLE);
					TEST_BUSY_CONDITION(HmiRecipe.Status.ProductRecipeLoaded == false);
					ActSubState = 2;
					break;

				case 2:
					TEST_BUSY_CONDITION(MpRecipeUIConnect.Status == mpRECIPE_UI_STATUS_REFRESH);
					ActSubState = 3;
					break;

				case 3:
					TEST_BUSY_CONDITION(MpRecipeUIConnect.Status != mpRECIPE_UI_STATUS_IDLE);
					TestState = TEST_ASSERT;
					break;
			}
			break;

		case TEST_ASSERT:
			TEST_ASSERT(RecipeExists("test.mcfg"));
			TEST_DONE;
			break;
	}
	TEST_BUSY;

}

_TEST CreateExisting(void)
{
	TIMEOUT_TEST_CASE
	switch (TestState)
	{
		case TEST_ARRANGE:
			strcpy(HmiRecipe.Parameters.FileName, "Machine");
			TEST_BUSY_CONDITION(MpRecipeUIConnect.Status != mpRECIPE_UI_STATUS_IDLE);
			TEST_BUSY_CONDITION(HmiRecipe.Status.HMIcommand != REC_HMI_WAIT);
			TestState = TEST_ACT;
			break;

		case TEST_ACT:
			TestState = TEST_ASSERT;
			break;

		case TEST_ASSERT:
			HmiRecipe.Commands.CreateRecipe = false;
			TEST_ASSERT(HmiRecipe.Status.FileDuplicate);
			TEST_ASSERT(RecipeExists("Machine.mcfg"));
			TEST_DONE;
			break;
	}
	TEST_BUSY;
}

_TEST CreateNonExisting(void)
{
	TIMEOUT_TEST_CASE
	switch (TestState)
	{
		case TEST_ARRANGE:
			strcpy(HmiRecipe.Parameters.FileName, "test2");
			TEST_BUSY_CONDITION(MpRecipeUIConnect.Status != mpRECIPE_UI_STATUS_IDLE);
			TEST_BUSY_CONDITION(HmiRecipe.Status.HMIcommand != REC_HMI_WAIT);
			TestState = TEST_ACT;
			break;

		case TEST_ACT:
			TestState = TEST_ASSERT;
			break;

		case TEST_ASSERT:
			HmiRecipe.Commands.CreateRecipe = false;
			TEST_ASSERT(!HmiRecipe.Status.FileDuplicate);
			TEST_ASSERT(!RecipeExists("test2.mcfg"));
			TEST_DONE;
			break;
	}
	TEST_BUSY;
}

_TEST CreateActive(void)
{
	TIMEOUT_TEST_CASE
	switch (TestState)
	{
		case TEST_ARRANGE:
			strcpy(HmiRecipe.Parameters.FileName, strtok(HmiRecipe.Status.LastLoadedConfigRecipe, "."));
			TEST_BUSY_CONDITION(MpRecipeUIConnect.Status != mpRECIPE_UI_STATUS_IDLE);
			TEST_BUSY_CONDITION(HmiRecipe.Status.HMIcommand != REC_HMI_WAIT);
			TestState = TEST_ACT;
			break;

		case TEST_ACT:
			TestState = TEST_ASSERT;
			break;

		case TEST_ASSERT:
			HmiRecipe.Commands.CreateRecipe = false;
			TEST_ASSERT(HmiRecipe.Status.FileDuplicate);
			TEST_ASSERT(RecipeExists(HmiRecipe.Status.LastLoadedConfigRecipe));
			TEST_DONE;
			break;
	}
	TEST_BUSY;
}

_TEST Preview(void)
{
	TIMEOUT_TEST_CASE
	switch (TestState)
	{
		case TEST_ARRANGE:
			MachineSettings.AddMachineSettingsHere1 = 157;
			MachineSettings.AddMachineSettingsHere2 = 43956;
			MachineSettings.AddMachineSettingsHere3 = true;
			MachineSettings.AddMachineSettingsHere4 = 134.876;
			MachineSettings.AddMachineSettingsHere5 = 4373;
			strcpy(HmiRecipe.Parameters.FileName, "preview");
			TEST_BUSY_CONDITION(MpRecipeUIConnect.Status != mpRECIPE_UI_STATUS_IDLE);
			TEST_BUSY_CONDITION(HmiRecipe.Status.HMIcommand != REC_HMI_WAIT);
			TestState = TEST_ACT;
			break;

		case TEST_ACT:
			if (MpRecipeUIConnect.Status == mpRECIPE_UI_STATUS_ERROR)
			{
				TEST_FAIL("MpRecipeUIConnect in error state");
				TEST_DONE;
			}
			switch (ActSubState)
			{
				case 0:
					HmiRecipe.Commands.CreateRecipe = true;
					TEST_BUSY_CONDITION(MpRecipeUIConnect.Status != mpRECIPE_UI_STATUS_CREATE);
					HmiRecipe.Commands.CreateRecipe = false;
					ActSubState = 1;
				break;

				case 1:
					TEST_BUSY_CONDITION(MpRecipeUIConnect.Status != mpRECIPE_UI_STATUS_IDLE);
					TEST_BUSY_CONDITION(HmiRecipe.Status.ProductRecipeLoaded == false);
					ActSubState = 2;
				break;

				case 2:
					TEST_BUSY_CONDITION(MpRecipeUIConnect.Status == mpRECIPE_UI_STATUS_REFRESH);
					ActSubState = 3;
				break;

				case 3:
					TEST_BUSY_CONDITION(MpRecipeUIConnect.Status != mpRECIPE_UI_STATUS_IDLE);
					TEST_BUSY_CONDITION(!SelectRecipe("preview.mcfg"));
					ActSubState = 4;
				break;

				case 4:
					TEST_BUSY_CONDITION(!SelectRecipe("preview.mcfg"));
					MpRecipeUIConnect.Recipe.Load = true;
					TEST_BUSY_CONDITION(MpRecipeUIConnect.Status != mpRECIPE_UI_STATUS_LOAD);
					MpRecipeUIConnect.Recipe.Load = false;
					ActSubState = 5;
				break;

				case 5:
					TEST_BUSY_CONDITION(MpRecipeUIConnect.Status != mpRECIPE_UI_STATUS_IDLE);
					TestState = TEST_ASSERT;
				break;
			}
			break;

		case TEST_ASSERT:
			TEST_ASSERT_EQUAL_INT(11, MachineSettings.AddMachineSettingsHere1);
			TEST_ASSERT_EQUAL_INT(22, MachineSettings.AddMachineSettingsHere2);
			TEST_ASSERT_EQUAL_INT(true, MachineSettings.AddMachineSettingsHere3);
			TEST_ASSERT_DOUBLE_WITHIN(0.0001, 3.2999999, MachineSettings.AddMachineSettingsHere4);
			TEST_ASSERT_EQUAL_INT(44, MachineSettings.AddMachineSettingsHere5);
			TEST_DONE;
			break;
	}
	TEST_BUSY;
}

_TEST Delete(void)
{
	TIMEOUT_TEST_CASE
	switch (TestState)
	{
		case TEST_ARRANGE:
			switch (ArrangeSubState)
			{
				case 0:
					strcpy(HmiRecipe.Parameters.FileName, "test");
					TEST_BUSY_CONDITION(MpRecipeUIConnect.Status != mpRECIPE_UI_STATUS_IDLE);
					TEST_BUSY_CONDITION(HmiRecipe.Status.HMIcommand != REC_HMI_WAIT);
					ArrangeSubState = 1;
					break;

				case 1:
					HmiRecipe.Commands.CreateRecipe = true;
					TEST_BUSY_CONDITION(MpRecipeUIConnect.Status != mpRECIPE_UI_STATUS_CREATE);
					HmiRecipe.Commands.CreateRecipe = false;
					ArrangeSubState = 2;
					break;

				case 2:
					TEST_BUSY_CONDITION(MpRecipeUIConnect.Status != mpRECIPE_UI_STATUS_IDLE);
					TEST_BUSY_CONDITION(HmiRecipe.Status.ProductRecipeLoaded == false);
					ArrangeSubState = 3;
					break;

				case 3:
					TEST_BUSY_CONDITION(MpRecipeUIConnect.Status == mpRECIPE_UI_STATUS_REFRESH);
					ArrangeSubState = 4;
					break;

				case 4:
					TEST_BUSY_CONDITION(MpRecipeUIConnect.Status != mpRECIPE_UI_STATUS_IDLE);
					ArrangeSubState = 5;
					break;

				case 5:
					TEST_BUSY_CONDITION(!SelectRecipe("test.mcfg"));
					TEST_BUSY_CONDITION(MpRecipeUIConnect.Status != mpRECIPE_UI_STATUS_IDLE);
					TEST_BUSY_CONDITION(HmiRecipe.Status.HMIcommand != REC_HMI_WAIT);
					TestState = TEST_ACT;
					break;
			}
			break;

		case TEST_ACT:
			if (MpRecipeUIConnect.Status == mpRECIPE_UI_STATUS_ERROR)
			{
				TEST_FAIL("MpRecipeUIConnect in error state");
				TEST_DONE;
			}
			switch (ActSubState)
			{
				case 0:
					MpRecipeUIConnect.Recipe.Delete = true;
					TEST_BUSY_CONDITION(MpRecipeUIConnect.MessageBox.LayerStatus != 0);
					MpRecipeUIConnect.Recipe.Delete = false;
					MpRecipeUIConnect.MessageBox.Confirm = true;
					ActSubState = 1;
					break;

				case 1:
					MpRecipeUIConnect.MessageBox.Confirm = false;
					TEST_BUSY_CONDITION(MpRecipeUIConnect.MessageBox.LayerStatus == 0)
					TEST_BUSY_CONDITION(MpRecipeUIConnect.Status == mpRECIPE_UI_STATUS_IDLE);
					ActSubState = 2;
					break;

				case 2:
					TEST_BUSY_CONDITION(MpRecipeUIConnect.Status != mpRECIPE_UI_STATUS_IDLE);
					ActSubState = 3;
					break;

				case 3:
					TEST_BUSY_CONDITION(MpRecipeUIConnect.Status == mpRECIPE_UI_STATUS_REFRESH);
					ActSubState = 4;
					break;

				case 4:
					TEST_BUSY_CONDITION(MpRecipeUIConnect.Status != mpRECIPE_UI_STATUS_IDLE);
					TestState = TEST_ASSERT;
					break;
			}
			break;

		case TEST_ASSERT:
			TEST_ASSERT(!RecipeExists("test.mcfg"));
			TEST_DONE;
			break;
	}
	TEST_BUSY;
}

_TEST Invalid(void)
{
	TIMEOUT_TEST_CASE
	switch (TestState)
	{
		case TEST_ARRANGE:
			switch (ArrangeSubState) {
				case 0:
					FileCopy_UT.enable = true;
					FileCopy_UT.pSrcDev = "mappRecipeFiles";
					FileCopy_UT.pSrc = "CSVformat\\Machine.mcfg";
					FileCopy_UT.pDestDev = "mappRecipeFiles";
					FileCopy_UT.pDest = "MachineInvalid.mcfg";
					FileCopy_UT.option= fiOVERWRITE;
					FileCopy(&FileCopy_UT);
					TEST_BUSY_CONDITION(FileCopy_UT.status == 65535);
					FileCopy_UT.enable = false;
					FileCopy(&FileCopy_UT);
					ArrangeSubState = 1;
					break;

				case 1:
					MpRecipeUIConnect.Recipe.Refresh = true;
					TEST_BUSY_CONDITION(MpRecipeUIConnect.Status == mpRECIPE_UI_STATUS_IDLE);
					MpRecipeUIConnect.Recipe.Refresh = false;
					ArrangeSubState = 2;
					break;

				case 2:
					TEST_BUSY_CONDITION(MpRecipeUIConnect.Status == mpRECIPE_UI_STATUS_REFRESH);
					ArrangeSubState = 3;
					break;

				case 3:
					TEST_BUSY_CONDITION(!SelectRecipe("MachineInvalid.mcfg"));
					TEST_BUSY_CONDITION(MpRecipeUIConnect.Status != mpRECIPE_UI_STATUS_IDLE);
					TEST_BUSY_CONDITION(HmiRecipe.Status.HMIcommand != REC_HMI_WAIT);
					TestState = TEST_ACT;
					break;
			}
			break;

		case TEST_ACT:
			switch (ActSubState)
			{
				case 0:
					MpRecipeUIConnect.Recipe.Load = true;
					TEST_BUSY_CONDITION(MpRecipeUIConnect.Status != mpRECIPE_UI_STATUS_LOAD);
					MpRecipeUIConnect.Recipe.Load = false;
					ActSubState = 1;
					break;

				case 1:
					TEST_BUSY_CONDITION(MpRecipeUIConnect.Status == mpRECIPE_UI_STATUS_LOAD);
					TestState = TEST_ASSERT;
					break;
			}
			break;

		case TEST_ASSERT:
			TEST_ASSERT_EQUAL_INT(mpRECIPE_UI_STATUS_ERROR, MpRecipeUIConnect.Status);
			TEST_DONE;
			break;
	}
	TEST_BUSY;
}

/*
B+R UnitTest: This is generated code.
Do not edit! Do not move!
Description: UnitTest Testprogramm infrastructure (TestSet).
LastUpdated: 2022-11-03 15:12:53Z
By B+R UnitTest Helper Version: 2.0.1.59
*/
UNITTEST_FIXTURES(fixtures)
{
	new_TestFixture("DefaultValues", DefaultValues),
	new_TestFixture("CreateNew", CreateNew),
	new_TestFixture("CreateExisting", CreateExisting),
	new_TestFixture("CreateNonExisting", CreateNonExisting),
	new_TestFixture("CreateActive", CreateActive),
	new_TestFixture("Preview", Preview),
	new_TestFixture("Delete", Delete),
	new_TestFixture("Invalid", Invalid),
};

UNITTEST_CALLER_COMPLETE_EXPLICIT(Set_RecipeMachineSettings, "Set_RecipeMachineSettings", setupTest, teardownTest, fixtures, setupSet, teardownSet, cyclicSetCaller);
```

#### Set_RecipeMgr.c - not listed in the package file held
```c
#include <bur/plctypes.h>

#ifdef _DEFAULT_INCLUDES
#include <AsDefault.h>
#endif

#include "UnitTest.h"
#include <stdbool.h>
#include <string.h>

_SETUP_SET(void)
{
	TEST_DONE;
}

_TEARDOWN_SET(void)
{
	TEST_DONE;
}

_SETUP_TEST(void)
{
    TEST_DONE;
}

_TEARDOWN_TEST(void)
{
	TEST_DONE;
}

/*
B+R UnitTest: This is generated code.
Do not edit! Do not move!
Description: UnitTest Testprogramm infrastructure (TestSet).
LastUpdated: 2022-09-22 12:42:06Z
By B+R UnitTest Helper Version: 2.0.1.59
*/
UNITTEST_FIXTURES(fixtures)
{
};

UNITTEST_CALLER_COMPLETE_EXPLICIT(Set_RecipeMgr, "Set_RecipeMgr", setupTest, teardownTest, fixtures, setupSet, teardownSet, 0);
```

### Package Logical/UnitTest/UserX - Package for mapp UserX Framework

### Program Logical/UnitTest/UserX/UserXUnitTest (ANSIC) - Unit Tests for UserX

- UserXMgr.typ (reference to Logical/Infrastructure/UserX/UserXMgr/UserXMgr.typ)

- UserXMgr.var (reference to Logical/Infrastructure/UserX/UserXMgr/UserXMgr.var)

#### variables.var - Name the suite and add PVs for the program
```iecst
(********************************************************************
 * COPYRIGHT --
 ********************************************************************
 * Program: utTemplate_automated
 * File: variables.var
 * Author: -
 * Created: -
 ********************************************************************
 * Local variables of program utTemplate_automated
 ********************************************************************)
(*Describe the test*)
VAR
	TestStep : USINT;
	Testsuite : UtMgrTestSuite := (Name:='UserMgr',Description:='UserMgr Unit Tests',MetaInformation:='Meta');
END_VAR
(*Variables used in the tests*)
VAR
	cycleCount : USINT;
	UT_Password : WSTRING[80] := "123ABc"; (*Unit test password login request*)
	UT_Username : WSTRING[80] := "Admin"; (*Unit test username login request *)
	UT_Compare : DINT; (*Unit test string compare PV holder*)
	UT_Message : STRING[80]; (*Unit test message variable*)
	UT_j : USINT; (*index for FOR loops*)
	UT_i : USINT; (*index for FOR loops*)
	UT_RoleList : ARRAY[0..4] OF WSTRING[50] := ["Administrators","Operators","Service",2("")]; (*Unit test role list for checking against user list*)
	UT_UserList : ARRAY[0..4] OF WSTRING[50] := ["Admin","Operator","Service_Tech",2("")]; (*Unit test user list for checking against user list*)
END_VAR
```

#### testSuite.c
```c
/********************************************************************
 * COPYRIGHT --
 ********************************************************************
 * Program: -
 * Author:
 * Created:
 ********************************************************************
 * Test registration and handshake
 ********************************************************************/

#include <bur/plctypes.h>

#ifdef _DEFAULT_INCLUDES
#include <AsDefault.h>
#endif
#include <string.h>

#include "UnitTest.h"

void _INIT initTestSuite(void)
{
    Testsuite.Enable = 1;
	utInit(&Testsuite);

    CommonTestsuite.Enable = 1;
    utInit(&CommonTestsuite);

    strcpy((char*)&FileDeviceName, "mappUserXFiles");
    strcpy((char*)&TextNameSpace, "mappFramework/UserX/Alarms");
    strcpy((char*)&TextID, "UserLocked");

}

void _CYCLIC cyclicWithTest(void)
{
	utCyclic(&Testsuite);
}

void _EXIT exitTestSuite(void)
{
	utExit(&Testsuite);
}
```

#### autoGeneratedFile.c - Auto generated code - list of all test sets in the program
```c
/*
B+R UnitTest: This is generated code.
Do not edit! Do not move!
Description: UnitTest Testprogramm infrastructure (List of TestSets).
LastUpdated: 2022-09-22 14:29:53Z
By B+R UnitTest Helper Version: 2.0.1.59
*/
#include "UnitTest.h"

UNITTEST_TESTSET_DECLARATION  Set_UserXMgr;
UNITTEST_TESTSET_DECLARATION  Set_Common;

UNITTEST_TESTSET_FIXTURES(utTestSets)
{
	new_TestSet(Set_UserXMgr),
	new_TestSet(Set_Common),
};
UNTITTEST_TESTSET_HANDLER();
```

#### Set_UserXMgr.c
```c
#include <bur/plctypes.h>

#ifdef _DEFAULT_INCLUDES
#include <AsDefault.h>
#endif

#include "UnitTest.h"
#include <stdbool.h>
#include <string.h>

_SETUP_SET(void)
{
	TEST_DONE;
}

_TEARDOWN_SET(void)
{
	TEST_DONE;
}

_SETUP_TEST(void)
{
//		TODO: Fix issue with variable mapping or removal of UserX MpUserXLogin_0 from framework as it is not used.
//	  switch (TestStep)
//	  {
//		  case 0:
//			  TEST_ABORT_CONDITION(MpUserXLogin_0.MpLink == 0);
//			  MpUserXLogin_0.Enable = 1;
//			  brwcscpy((UDINT)&UT_Username, (UDINT)&UT_UserList[0]);
//			  MpUserXLogin_0.UserName = (UDINT)&UT_Username;
//			  MpUserXLogin_0.Password = (UDINT)&UT_Password;
//			  MpUserXLogin_0.Login = 1;
//			  MpUserXLogin(&MpUserXLogin_0);
//			  UT_Compare = brwcscmp((UDINT)&MpUserXLogin_0.CurrentUser, (UDINT)&UT_Username);
//			  TEST_BUSY_CONDITION(UT_Compare != 0);
//			  if (UT_Compare == 0){
//				  TEST_ABORT_CONDITION(UserXLoginUIConnect.Status == mpUSERX_UI_STATUS_ERROR);
//				  MpUserXLogin_0.Login = 0;
//				  TestStep = 1;
//			  }
//			  break;
//		  case 1:
//			  UT_Compare = brwcscmp((UDINT)&MpUserXLogin_0.CurrentUser, (UDINT)&UT_Username);
//			  TEST_ABORT_CONDITION(UT_Compare != 0);
//			  TestStep = 0;
//			  TEST_DONE;
//			  break;
//	  }
//	  TEST_BUSY;
	TEST_DONE; // Temporary
}

_TEST USERX_ROLES_CHECK(void)
{
//		See Note in setup
//	  switch (TestStep){
//		  case 0:
//			  UT_Compare = brwcscmp((UDINT)&MpUserXLogin_0.CurrentUser, (UDINT)&UT_Username);
//			  TEST_ABORT_CONDITION(UT_Compare != 0); // Check to make sure role is admin so all users / roles can be seen
//			  for (UT_i = 0; UT_i < (sizeof(UT_RoleList) / sizeof(UT_RoleList[0]) - 1); UT_i++)
//			  {
//				  for (UT_j = 0; UT_j < (sizeof(UserXMgrUIConnect.Role.List.Names) / sizeof(UserXMgrUIConnect.Role.List.Names[0]) - 1); UT_j++)
//				  {
//					  UT_Compare = brwcscmp((UDINT)&UserXMgrUIConnect.Role.List.Names[UT_j], (UDINT)&UT_RoleList[UT_i]);
//					  if (UT_Compare == 0)
//					  {
//
//						  break;
//					  }
//				  }
//				  if (UT_RoleList[UT_i] != "")
//				  {
//					  TEST_ASSERT(UT_Compare == 0);
//				  }
//			  }
//			  TestStep = 1;
//			  break;
//		  case 1:
//			  TestStep = 0;
//			  TEST_DONE;
//			  break;
//	  }
//	  TEST_BUSY;
	TEST_DONE; // Temporary
}

_TEST USERX_USER_CHECK(void)
{
//		See Note in setup
//
//	  switch (TestStep){
//		  case 0: // Ensure Admin has Admin Role
//			  UT_Compare = brwcscmp((UDINT)&MpUserXLogin_0.CurrentUser, (UDINT)&UT_Username);
//			  TEST_ABORT_CONDITION(UT_Compare != 0);
//			  TEST_ABORT_CONDITION(MpUserXLogin_0.MpLink == 0);
//			  TestStep = 1;
//			  break;
//		  case 1:
//			  TEST_ABORT_CONDITION(MpUserXLogin_0.MpLink == 0);
//			  brwcscpy((UDINT)&UT_Username, (UDINT)&UT_UserList[1]);
//			  MpUserXLogin_0.Enable = 1;
//			  MpUserXLogin_0.UserName = (UDINT)&UT_Username;
//			  MpUserXLogin_0.Password = (UDINT)&UT_Password;
//			  MpUserXLogin_0.Login = 1;
//			  MpUserXLogin(&MpUserXLogin_0);
//			  while (MpUserXLogin_0.CommandBusy == 1){
//				  MpUserXLogin(&MpUserXLogin_0);
//			  }
//			  UT_Compare = brwcscmp((UDINT)&MpUserXLogin_0.CurrentUser, (UDINT)&UT_Username);
//			  TEST_ASSERT(UT_Compare == 0);
//			  if (UT_Compare == 0){
//				  MpUserXLogin_0.Login = 0;
//				  //	TODO: UIConnect does not update on user change this may require that the password be reset as required by the configuration
//				  //UT_Compare = brwcscmp((UDINT)&UT_RoleList[1], (UDINT)&UserXMgrUIConnect.Role.Info.Name);
//				  //TEST_ASSERT(UT_Compare == 0);
//				  TestStep = 2;
//			  }
//			  break;
//
//		  case 2:
//			  TEST_ABORT_CONDITION(MpUserXLogin_0.MpLink == 0);
//			  brwcscpy((UDINT)&UT_Username, (UDINT)&UT_UserList[2]);
//			  MpUserXLogin_0.Enable = 1;
//			  MpUserXLogin_0.UserName = (UDINT)&UT_Username;
//			  MpUserXLogin_0.Password = (UDINT)&UT_Password;
//			  MpUserXLogin_0.Login = 1;
//			  MpUserXLogin(&MpUserXLogin_0);
//			  while (MpUserXLogin_0.CommandBusy == 1){
//				  MpUserXLogin(&MpUserXLogin_0);
//			  }
//			  UT_Compare = brwcscmp((UDINT)&MpUserXLogin_0.CurrentUser, (UDINT)&UT_Username);
//			  TEST_ASSERT(UT_Compare == 0);
//			  if (UT_Compare == 0){
//				  MpUserXLogin_0.Login = 0;
////				TODO: UIConnect does not update on user change this may require that the password be reset as required by the configuration
////				UT_Compare = brwcscmp((UDINT)&UT_RoleList[2], (UDINT)&UserXMgrUIConnect.Role.Info.Name);
////				TEST_ASSERT(UT_Compare == 0);
//				  TestStep = 3;
//			  }
//			  break;
//		  case 3:
//			  TEST_ABORT_CONDITION(MpUserXLogin_0.MpLink == 0);
//			  brwcscpy((UDINT)&UT_Username, (UDINT)&UT_UserList[0]);
//			  MpUserXLogin_0.Enable = 1;
//			  MpUserXLogin_0.UserName = (UDINT)&UT_Username;
//			  MpUserXLogin_0.Password = (UDINT)&UT_Password;
//			  MpUserXLogin_0.Login = 1;
//			  MpUserXLogin(&MpUserXLogin_0);
//			  while (MpUserXLogin_0.CommandBusy == 1){
//				  MpUserXLogin(&MpUserXLogin_0);
//			  }
//			  UT_Compare = brwcscmp((UDINT)&MpUserXLogin_0.CurrentUser, (UDINT)&UT_Username);
//			  TEST_ASSERT(UT_Compare == 0);
//			  if (UT_Compare == 0){
//				  MpUserXLogin_0.Login = 0;
//				  TestStep = 4;
//			  }
//			  break;
//		  case 4:
//			  TestStep = 0;
//			  TEST_DONE;
//			  break;
//	  }
//	  TEST_BUSY;
	TEST_DONE; // Temporary
}

_TEST USERX_LOGOUT(void){
	//		See Note in setup
//	  switch (TestStep){
//		  case 0:
//			  TEST_ABORT_CONDITION(MpUserXLogin_0.MpLink == 0);
//			  MpUserXLogin_0.Enable = 1;
//			  MpUserXLogin_0.Logout = 1;
//			  MpUserXLogin(&MpUserXLogin_0);
//			  while (MpUserXLogin_0.CommandBusy == 1){
//				  MpUserXLogin(&MpUserXLogin_0);
//			  }
//			  TestStep = 1;
//			  break;
//		  case 1:
//			  TEST_ASSERT(MpUserXLogin_0.CurrentLevel != 0);
//			  TestStep = 2;
//			  break;
//		  case 2:
//			  TestStep = 0;
//			  TEST_DONE;
//			  break;
//	  }
	TEST_DONE; // Temporary
}
_TEARDOWN_TEST(void)
{
	TEST_DONE;
}

/*
B+R UnitTest: This is generated code.
Do not edit! Do not move!
Description: UnitTest Testprogramm infrastructure (TestSet).
LastUpdated: 2022-11-09 20:10:20Z
By B+R UnitTest Helper Version: 2.0.1.59
*/
UNITTEST_FIXTURES(fixtures)
{
	new_TestFixture("USERX_ROLES_CHECK", USERX_ROLES_CHECK),
	new_TestFixture("USERX_USER_CHECK", USERX_USER_CHECK),
	new_TestFixture("USERX_LOGOUT", USERX_LOGOUT),
};

UNITTEST_CALLER_COMPLETE_EXPLICIT(Set_UserXMgr, "Set_UserXMgr", setupTest, teardownTest, fixtures, setupSet, teardownSet, 0);
```

- CommonVariables.var (reference to Logical/UnitTest/Common/CommonUT/CommonVariables.var)

- Set_Common.c (reference to Logical/UnitTest/Common/CommonUT/Set_Common.c)

### Package Logical/UnitTest/Report - Package for mapp Report Framework

### Program Logical/UnitTest/Report/ReportUnitTest (ANSIC)

- ReportMgr.typ (reference to Logical/Infrastructure/Report/ReportMgr/ReportMgr.typ)

- ReportMgr.var (reference to Logical/Infrastructure/Report/ReportMgr/ReportMgr.var)

#### testSuite.c
```c
/********************************************************************
 * COPYRIGHT --
 ********************************************************************
 * Program: -
 * Author:
 * Created:
 ********************************************************************
 * Test registration and handshake
 ********************************************************************/

#include <bur/plctypes.h>

#ifdef _DEFAULT_INCLUDES
#include <AsDefault.h>
#endif

#include "UnitTest.h"
#include <string.h>

void _INIT initTestSuite(void)
{
    Testsuite.Enable = 1;
	utInit(&Testsuite);

    CommonTestsuite.Enable = 1;
    utInit(&CommonTestsuite);

    strcpy((char*)&FileDeviceName, "mappReportFiles");
    strcpy((char*)&TextNameSpace, "mappFramework/Report/Alarms");
    strcpy((char*)&TextID, "GenerateFailed");

}

void _CYCLIC cyclicWithTest(void)
{
	utCyclic(&Testsuite);
}

void _EXIT exitTestSuite(void)
{
	utExit(&Testsuite);
}
```

#### autoGeneratedFile.c - Auto generated code - list of all test sets in the program
```c
/*
B+R UnitTest: This is generated code.
Do not edit! Do not move!
Description: UnitTest Testprogramm infrastructure (List of TestSets).
LastUpdated: 2022-11-14 19:41:10Z
By B+R UnitTest Helper Version: 2.0.1.59
*/
#include "UnitTest.h"

UNITTEST_TESTSET_DECLARATION  Set_ReportMgr;
UNITTEST_TESTSET_DECLARATION  Set_Common;

UNITTEST_TESTSET_FIXTURES(utTestSets)
{
	new_TestSet(Set_ReportMgr),
	new_TestSet(Set_Common),
};
UNTITTEST_TESTSET_HANDLER();
```

#### Set_ReportMgr.c
```c
#include <bur/plctypes.h>

#ifdef _DEFAULT_INCLUDES
#include <AsDefault.h>
#endif

#include "UnitTest.h"
#include <stdbool.h>
#include <string.h>

_SETUP_SET(void)
{
	TEST_DONE;
}

_TEARDOWN_SET(void)
{
	TEST_DONE;
}

_SETUP_TEST(void)
{
    TEST_DONE;
}

_TEARDOWN_TEST(void)
{
	TEST_DONE;
}

_TEST CreateAdvReport(void)
{
    switch (TestState)
    {
        case TEST_ARRANGE:
         	HmiReport_UT.Parameters.UseAdvancedFormat = true;
			TEST_BUSY_CONDITION(CoreInfoActive == true);
            TEST_ABORT_CONDITION(HmiReport_UT.Status.Error == true);
            TestState = TEST_ACT;
            break;

        case TEST_ACT:
			TEST_BUSY_CONDITION(CoreInfoActive == false);
			HmiReport_UT.Commands.Generate = true;
			TEST_BUSY_CONDITION(HmiReport_UT.Status.Busy == false);
            TestState = TEST_ASSERT;
            break;

        case TEST_ASSERT:
            HmiReport_UT.Commands.Generate = false;
			TEST_BUSY_CONDITION(HmiReport_UT.Status.Busy == true);
            TEST_ASSERT(HmiReport_UT.Status.Error == false);
			TEST_ASSERT_EQUAL_INT(1, CoreInfo_UT.NumberOfReports);
            TEST_DONE;
            break;
    }
    TEST_BUSY;
}

_TEST CreateSimpleReport(void)
{
    switch (TestState)
    {
        case TEST_ARRANGE:
         	HmiReport_UT.Parameters.UseAdvancedFormat = false;
			TEST_BUSY_CONDITION(CoreInfoActive == true);
            TEST_ABORT_CONDITION(HmiReport_UT.Status.Error == true);
            TestState = TEST_ACT;
            break;

        case TEST_ACT:
			TEST_BUSY_CONDITION(CoreInfoActive == false);
			HmiReport_UT.Commands.Generate = true;
			TEST_BUSY_CONDITION(HmiReport_UT.Status.Busy == false);
            TestState = TEST_ASSERT;
            break;

        case TEST_ASSERT:
            HmiReport_UT.Commands.Generate = false;
			TEST_BUSY_CONDITION(HmiReport_UT.Status.Busy == true);
            TEST_ASSERT(HmiReport_UT.Status.Error == false);
			TEST_ASSERT_EQUAL_INT(1, CoreInfo_UT.NumberOfReports);
            TEST_DONE;
            break;
    }
    TEST_BUSY;
}

/*
B+R UnitTest: This is generated code.
Do not edit! Do not move!
Description: UnitTest Testprogramm infrastructure (TestSet).
LastUpdated: 2022-11-15 21:58:19Z
By B+R UnitTest Helper Version: 2.0.1.59
*/
UNITTEST_FIXTURES(fixtures)
{
	new_TestFixture("CreateAdvReport", CreateAdvReport),
	new_TestFixture("CreateSimpleReport", CreateSimpleReport),
};

UNITTEST_CALLER_COMPLETE_EXPLICIT(Set_ReportMgr, "Set_ReportMgr", setupTest, teardownTest, fixtures, setupSet, teardownSet, 0);
```

- CommonVariables.var (reference to Logical/UnitTest/Common/CommonUT/CommonVariables.var)

- Set_Common.c (reference to Logical/UnitTest/Common/CommonUT/Set_Common.c)

### Program Logical/UnitTest/Common/CommonUT (ANSIC) - Unit Tests for FileMgr

- CommonVariables.var (reference to Logical/UnitTest/Common/CommonUT/CommonVariables.var)

#### testSuite.c
```c
/********************************************************************
 * COPYRIGHT --
 ********************************************************************
 * Program: -
 * Author:
 * Created:
 ********************************************************************
 * Test registration and handshake
 ********************************************************************/

#include <bur/plctypes.h>

#ifdef _DEFAULT_INCLUDES
#include <AsDefault.h>
#endif

#include "UnitTest.h"

void _INIT initTestSuite(void)
{
    Testsuite.Enable = 1;
	utInit(&Testsuite);
}

void _CYCLIC cyclicWithTest(void)
{
	utCyclic(&Testsuite);
}

void _EXIT exitTestSuite(void)
{
	utExit(&Testsuite);
}
```

#### autoGeneratedFile.c - Auto generated code - list of all test sets in the program
```c
/*
B+R UnitTest: This is generated code.
Do not edit! Do not move!
Description: UnitTest Testprogramm infrastructure (List of TestSets).
LastUpdated: 2022-09-22 11:55:24Z
By B+R UnitTest Helper Version: 2.0.1.59
*/
#include "UnitTest.h"

UNITTEST_TESTSET_DECLARATION  Set_Common;

UNITTEST_TESTSET_FIXTURES(utTestSets)
{
	new_TestSet(Set_Common),
};
UNTITTEST_TESTSET_HANDLER();
```

- Set_Common.c (reference to Logical/UnitTest/Common/CommonUT/Set_Common.c)

- Update_TestPrograms_in_current_location.bat - Updates test programs within the current package (not shown)

### Package Logical/UnitTestVC4/AlarmX - Package for mapp AlarmX Framework

### Program Logical/UnitTestVC4/AlarmX/AlarmXUnitTest (ANSIC)

- AlarmMgr.typ (reference to Logical/Infrastructure/VC4/AlarmX/AlarmMgr/AlarmMgr.typ)

- AlarmMgr.var (reference to Logical/Infrastructure/VC4/AlarmX/AlarmMgr/AlarmMgr.var)

#### variables.var - Name the suite and add PVs for the program
```iecst
(********************************************************************
 * COPYRIGHT --
 ********************************************************************
 * Program: utTemplate_automated
 * File: variables.var
 * Author: -
 * Created: -
 ********************************************************************
 * Local variables of program utTemplate_automated
 ********************************************************************)
(*Describe the test*)
VAR
	Testsuite : UtMgrTestSuite := (Name:='AlarmMgrVC4',Description:='AlarmMgr VC4 Unit Tests',MetaInformation:='Meta');
END_VAR
(*Variables used in the tests*)
VAR
	MpAlarmXAcknowledgeAll_0 : MpAlarmXAcknowledgeAll;
	StartingActiveAlarms : UDINT;
	StartingPendingAlarms : UDINT;
	cycleCount : USINT;
END_VAR
```

#### testSuite.c
```c
/********************************************************************
 * COPYRIGHT --
 ********************************************************************
 * Program: -
 * Author:
 * Created:
 ********************************************************************
 * Test registration and handshake
 ********************************************************************/

#include <bur/plctypes.h>

#ifdef _DEFAULT_INCLUDES
#include <AsDefault.h>
#endif

#include "UnitTest.h"
#include <string.h>
#include <stdbool.h>

void _INIT initTestSuite(void)
{
	Testsuite.Enable = 1;
	utInit(&Testsuite);

	CommonTestsuite.Enable = 1;
	utInit(&CommonTestsuite);

	strcpy((char*)&FileDeviceName, "mappAlarmXFiles");
	strcpy((char*)&TextNameSpace, "mappFramework/AlarmX/Alarms");
	strcpy((char*)&TextID, "EmergencyStop.0");
}

void _CYCLIC cyclicWithTest(void)
{
	utCyclic(&Testsuite);
}

void _EXIT exitTestSuite(void)
{
	utExit(&Testsuite);
}
```

#### autoGeneratedFile.c - Auto generated code - list of all test sets in the program
```c
/*
B+R UnitTest: This is generated code.
Do not edit! Do not move!
Description: UnitTest Testprogramm infrastructure (List of TestSets).
LastUpdated: 2022-11-23 14:37:56Z
By B+R UnitTest Helper Version: 2.0.1.59
*/
#include "UnitTest.h"

UNITTEST_TESTSET_DECLARATION  Set_AlarmExamples;
UNITTEST_TESTSET_DECLARATION  Set_AlarmMgr;
UNITTEST_TESTSET_DECLARATION  Set_Common;

UNITTEST_TESTSET_FIXTURES(utTestSets)
{
	new_TestSet(Set_AlarmExamples),
	new_TestSet(Set_AlarmMgr),
	new_TestSet(Set_Common),
};
UNTITTEST_TESTSET_HANDLER();
```

#### Set_AlarmExamples.c
```c
#include <bur/plctypes.h>

#ifdef _DEFAULT_INCLUDES
#include <AsDefault.h>
#endif

#include "UnitTest.h"
#include <stdbool.h>
#include <string.h>

#define _RESET_ALARMS																\
	AlarmExamples.LevelMonitoring = 50;												\
	MpAlarmXAcknowledgeAll_0.Execute = true;										\
	MpAlarmXAcknowledgeAll(&MpAlarmXAcknowledgeAll_0);								\
	TEST_BUSY_CONDITION(MpAlarmXAcknowledgeAll_0.CommandDone == false);				\
	MpAlarmXAcknowledgeAll_0.Execute = false;										\
	TEST_BUSY_CONDITION(MpAlarmXAcknowledgeAll_0.Info.UnacknowledgedAlarms != 0);	\
	TEST_BUSY_CONDITION(cycleCount < 25);

_SETUP_SET(void)
{
	_RESET_ALARMS;
	TEST_DONE;
}

_TEARDOWN_SET(void)
{
	_RESET_ALARMS;
	TEST_DONE;
}

_SETUP_TEST(void)
{
	cycleCount = 0;
	TEST_DONE;
}

_CYCLIC_SET(void)
{
	MpAlarmXAcknowledgeAll_0.MpLink = &gMpLinkAlarmXCore;
	MpAlarmXAcknowledgeAll_0.Enable = true;
	MpAlarmXAcknowledgeAll(&MpAlarmXAcknowledgeAll_0);

	cycleCount++;

	TEST_ABORT_CONDITION(cycleCount == 254);
}

bool AlarmIsActive(char* alarmName)
{
	for (USINT i = 0; i < (sizeof(MpAlarmXListUIConnect.AlarmList.Name)/sizeof(MpAlarmXListUIConnect.AlarmList.Name[0])); i++)
	{
		if ((strcmp(alarmName, MpAlarmXListUIConnect.AlarmList.Name[i]) == 0) && (MpAlarmXListUIConnect.AlarmList.StateActive[i] == true))
			return true;
	}
	return false;
}

void LogActiveAlarms(void)
{
	for (USINT i = 0; i < (sizeof(MpAlarmXListUIConnect.AlarmList.Name)/sizeof(MpAlarmXListUIConnect.AlarmList.Name[0])); i++)
	{
		if (strcmp(&"", MpAlarmXListUIConnect.AlarmList.Name[i]) != 0)
		{
			TEST_INFO(MpAlarmXListUIConnect.AlarmList.Name[i])
		}
	}
}

// These tests must run sequentially, Arrange->Act->Assert
// 3 "_TEST" function for each unit test
_TEST Arrange_LevelMonitoringLow(void)
{
	StartingActiveAlarms = MpAlarmXCoreMain.ActiveAlarms;
	StartingPendingAlarms = MpAlarmXCoreMain.PendingAlarms;
	_RESET_ALARMS;
	TEST_DONE;
}

_TEST Act_LevelMonitoringLow(void)
{
	AlarmExamples.LevelMonitoring = 19;
	TEST_BUSY_CONDITION(cycleCount < 10);
	TEST_DONE;
}

_TEST Assert_LevelMonitoringLow(void)
{
	TEST_ASSERT_MESSAGE(MpAlarmXCoreMain.PendingAlarms > StartingPendingAlarms, "Pending Alarms did not increase");
	TEST_ASSERT_MESSAGE(MpAlarmXCoreMain.ActiveAlarms > StartingActiveAlarms, "Active Alarms did not increase");
	TEST_ASSERT(AlarmIsActive("LevelMonitoringExample"));
	LogActiveAlarms();
	TEST_DONE;
}

_TEST Arrange_LevelMonitoringLowLow(void)
{
	StartingActiveAlarms = MpAlarmXCoreMain.ActiveAlarms;
	StartingPendingAlarms = MpAlarmXCoreMain.PendingAlarms;
	_RESET_ALARMS;
	TEST_DONE;
}

_TEST Act_LevelMonitoringLowLow(void)
{
	AlarmExamples.LevelMonitoring = 9;
	TEST_BUSY_CONDITION(cycleCount < 15);
	TEST_DONE;
}

_TEST Assert_LevelMonitoringLowLow(void)
{
	TEST_ASSERT_MESSAGE(MpAlarmXCoreMain.PendingAlarms > StartingPendingAlarms, "Pending Alarms did not increase");
	TEST_ASSERT_MESSAGE(MpAlarmXCoreMain.ActiveAlarms > StartingActiveAlarms, "Active Alarms did not increase");
	TEST_ASSERT(AlarmIsActive("LevelMonitoringExample"));
	LogActiveAlarms();
	TEST_DONE;
}

_TEST Arrange_LevelMonitoringHigh(void)
{
	StartingActiveAlarms = MpAlarmXCoreMain.ActiveAlarms;
	StartingPendingAlarms = MpAlarmXCoreMain.PendingAlarms;
	_RESET_ALARMS;
	TEST_DONE;
}

_TEST Act_LevelMonitoringHigh(void)
{
	AlarmExamples.LevelMonitoring = 81;
	TEST_BUSY_CONDITION(cycleCount < 15);
	TEST_DONE;
}

_TEST Assert_LevelMonitoringHigh(void)
{
	TEST_ASSERT_MESSAGE(MpAlarmXCoreMain.PendingAlarms > StartingPendingAlarms, "Pending Alarms did not increase");
	TEST_ASSERT_MESSAGE(MpAlarmXCoreMain.ActiveAlarms > StartingActiveAlarms, "Active Alarms did not increase");
	TEST_ASSERT(AlarmIsActive("LevelMonitoringExample"));
	LogActiveAlarms();
	TEST_DONE;
}

_TEST Arrange_LevelMonitoringHighHigh(void)
{
	StartingActiveAlarms = MpAlarmXCoreMain.ActiveAlarms;
	StartingPendingAlarms = MpAlarmXCoreMain.PendingAlarms;
	_RESET_ALARMS;
	TEST_DONE;
}

_TEST Act_LevelMonitoringHighHigh(void)
{
	AlarmExamples.LevelMonitoring = 91;
	TEST_BUSY_CONDITION(cycleCount < 15);
	TEST_DONE;
}

_TEST Assert_LevelMonitoringHighHigh(void)
{
	TEST_ASSERT_MESSAGE(MpAlarmXCoreMain.PendingAlarms > StartingPendingAlarms, "Pending Alarms did not increase");
	TEST_ASSERT_MESSAGE(MpAlarmXCoreMain.ActiveAlarms > StartingActiveAlarms, "Active Alarms did not increase");
	TEST_ASSERT(AlarmIsActive("LevelMonitoringExample"));
	LogActiveAlarms();
	TEST_DONE;
}

/*
B+R UnitTest: This is generated code.
Do not edit! Do not move!
Description: UnitTest Testprogramm infrastructure (TestSet).
LastUpdated: 2022-11-03 17:18:35Z
By B+R UnitTest Helper Version: 2.0.1.59
*/
UNITTEST_FIXTURES(fixtures)
{
	new_TestFixture("Arrange_LevelMonitoringLow", Arrange_LevelMonitoringLow),
	new_TestFixture("Act_LevelMonitoringLow", Act_LevelMonitoringLow),
	new_TestFixture("Assert_LevelMonitoringLow", Assert_LevelMonitoringLow),
	new_TestFixture("Arrange_LevelMonitoringLowLow", Arrange_LevelMonitoringLowLow),
	new_TestFixture("Act_LevelMonitoringLowLow", Act_LevelMonitoringLowLow),
	new_TestFixture("Assert_LevelMonitoringLowLow", Assert_LevelMonitoringLowLow),
	new_TestFixture("Arrange_LevelMonitoringHigh", Arrange_LevelMonitoringHigh),
	new_TestFixture("Act_LevelMonitoringHigh", Act_LevelMonitoringHigh),
	new_TestFixture("Assert_LevelMonitoringHigh", Assert_LevelMonitoringHigh),
	new_TestFixture("Arrange_LevelMonitoringHighHigh", Arrange_LevelMonitoringHighHigh),
	new_TestFixture("Act_LevelMonitoringHighHigh", Act_LevelMonitoringHighHigh),
	new_TestFixture("Assert_LevelMonitoringHighHigh", Assert_LevelMonitoringHighHigh),
};

UNITTEST_CALLER_COMPLETE_EXPLICIT(Set_AlarmExamples, "Set_AlarmExamples", setupTest, 0, fixtures, setupSet, teardownSet, cyclicSetCaller);
```

#### Set_AlarmMgr.c
```c
#include <bur/plctypes.h>

#ifdef _DEFAULT_INCLUDES
#include <AsDefault.h>
#endif

#include "UnitTest.h"
#include <stdbool.h>
#include <string.h>

_SETUP_SET(void)
{
	TEST_DONE;
}

_TEARDOWN_SET(void)
{
	TEST_DONE;
}

_SETUP_TEST(void)
{
    TEST_DONE;
}

_TEARDOWN_TEST(void)
{
	TEST_DONE;
}

_TEST CheckCommissioningModeActive(void)
{
	CommissioningModeActive = true;
	TEST_ASSERT(Alarms[0] == false);
}

/*
B+R UnitTest: This is generated code.
Do not edit! Do not move!
Description: UnitTest Testprogramm infrastructure (TestSet).
LastUpdated: 2023-01-30 14:31:38Z
By B+R UnitTest Helper Version: 2.0.1.59
*/
UNITTEST_FIXTURES(fixtures)
{
	new_TestFixture("CheckCommissioningModeActive", CheckCommissioningModeActive),
};

UNITTEST_CALLER_COMPLETE_EXPLICIT(Set_AlarmMgr, "Set_AlarmMgr", setupTest, teardownTest, fixtures, setupSet, teardownSet, 0);
```

#### Set_Common.c
```c
#include <bur/plctypes.h>

#ifdef _DEFAULT_INCLUDES
#include <AsDefault.h>
#endif

#include "UnitTest.h"
#include <stdbool.h>
#include <string.h>

_SETUP_SET(void)
{
	TEST_DONE;
}

_TEARDOWN_SET(void)
{
	TEST_DONE;
}

_SETUP_TEST(void)
{
	TEST_DONE;
}

_TEARDOWN_TEST(void)
{

	TEST_DONE;
}

_TEST FileDeviceExists(void)
{
	if (strcmp((char*)&FileDeviceName, "") == 0)
	{
		TEST_INFO_POS("FileDeviceName is empty");
		TEST_DONE;
	}
	DirInfoCommon_UT.enable = true;
	DirInfoCommon_UT.pDevice = (UDINT)&FileDeviceName;
	DirInfoCommon_UT.pPath = (UDINT)&"";
	DirInfo(&DirInfoCommon_UT);
	TEST_BUSY_CONDITION(DirInfoCommon_UT.status == 65535);
	TEST_ASSERT_EQUAL_INT(0, DirInfoCommon_UT.status);
	TEST_DONE;
}

_TEST NoFunctionBlockErrors(void)
{

	for (USINT i=0; i<(sizeof(MpBlockStatus)/sizeof(MpBlockStatus[0]));i++)
	{
		TEST_ASSERT_EQUAL_INT(0, MpBlockStatus[i]);
	}
	TEST_DONE;
}

_TEST TextFileConfirmation(void)
{
	// Arrange
	TEST_ABORT_CONDITION(strcmp(TextNameSpace, "") == 0);
	TEST_ABORT_CONDITION(strcmp(TextID, "") == 0);

	ArTextSysGetTextComon_UT.Execute = true;
	ArTextSysGetTextComon_UT.Namespace = (UDINT)&TextNameSpace;
	ArTextSysGetTextComon_UT.TextID = (UDINT)&TextID;
	strcpy((char*)&ArTextSysGetTextComon_UT.LanguageCode, "en");
	ArTextSysGetTextComon_UT.TextBuffer = (UDINT)&Text;
	ArTextSysGetTextComon_UT.TextBufferSize = sizeof(Text)/sizeof(Text[0]);

	// Act
	ArTextSysGetText(&ArTextSysGetTextComon_UT);
	TEST_BUSY_CONDITION(ArTextSysGetTextComon_UT.Busy);

	// Assert
	TEST_ASSERT(ArTextSysGetTextComon_UT.Error == false);
	TEST_ASSERT_EQUAL_INT(0, ArTextSysGetTextComon_UT.StatusID);
	TEST_ASSERT_MESSAGE(strcmp(Text, "") != 0, "Text is empty");
	TEST_DONE;
}

/*
B+R UnitTest: This is generated code.
Do not edit! Do not move!
Description: UnitTest Testprogramm infrastructure (TestSet).
LastUpdated: 2022-09-22 14:29:52Z
By B+R UnitTest Helper Version: 2.0.1.59
*/
UNITTEST_FIXTURES(fixtures)
{
	new_TestFixture("FileDeviceExists", FileDeviceExists),
	new_TestFixture("NoFunctionBlockErrors", NoFunctionBlockErrors),
	new_TestFixture("TextFileConfirmation", TextFileConfirmation),
};

UNITTEST_CALLER_COMPLETE_EXPLICIT(Set_Common, "Set_Common", setupTest, teardownTest, fixtures, setupSet, teardownSet, 0);
```

### Package Logical/UnitTestVC4/Audit - Package for mapp AlarmX Framework

### Program Logical/UnitTestVC4/Audit/AuditTest (ANSIC)

- AuditMgr.typ (reference to Logical/Infrastructure/VC4/Audit/AuditMgr/AuditMgr.typ)

- AuditMgr.var (reference to Logical/Infrastructure/VC4/Audit/AuditMgr/AuditMgr.var)

#### variables.var - Name the suite and add PVs for the program
```iecst
(********************************************************************
 * COPYRIGHT --
 ********************************************************************
 * Program: utTemplate_automated
 * File: variables.var
 * Author: -
 * Created: -
 ********************************************************************
 * Local variables of program utTemplate_automated
 ********************************************************************)
(*Describe the test*)
VAR
	Testsuite : UtMgrTestSuite := (Name:='AuditMgrVC4',Description:='AuditMgr VC4 Unit Tests',MetaInformation:='Meta');
END_VAR
(*Variables used in the tests*)
VAR
	cycleCount : {REDUND_UNREPLICABLE} UINT;
	SampleTemperature : REAL;
	DirInfo_0 : DirInfo;
	TestComparisonNumber : USINT;
	ActDelay : USINT;
	ArrangeDelay : USINT;
	AssertDelay : USINT;
	DTSetTime_0 : DTSetTime;
	HOUR : USINT := 16;
	MINUTE : USINT := 0;
	SET_TIME : DATE_AND_TIME := DT#2023-01-01-15:59:59;
	MAX_FILE_SIZE : UDINT := 100; (*Maximum file size for automatic archiving (Kb)*)
	SAMPLE_TEMP_VALUE : REAL := 5;
	DEFAULT_TEMP_VALUE : REAL := 6;
	TON_0 : TON;
	TIMER_LENGTH : TIME := T#2s;
	MpAuditTrailCmdDone : BOOL;
	MpAuditTrailError : BOOL;
	DelayCycles : USINT := 10;
END_VAR
```

#### testSuite.c
```c
/********************************************************************
 * COPYRIGHT --
 ********************************************************************
 * Program: -
 * Author:
 * Created:
 ********************************************************************
 * Test registration and handshake
 ********************************************************************/

#include <bur/plctypes.h>

#ifdef _DEFAULT_INCLUDES
#include <AsDefault.h>
#endif

#include "UnitTest.h"
#include <string.h>

void _INIT initTestSuite(void)
{
	Testsuite.Enable = 1;
	utInit(&Testsuite);

	CommonTestsuite.Enable = 1;
	utInit(&CommonTestsuite);

	strcpy((char*)&FileDeviceName, "mappAuditFiles");
	strcpy((char*)&TextNameSpace, "mappFramework/Audit/Alarms");
	strcpy((char*)&TextID, "ArchiveAvailable");
}

void _CYCLIC cyclicWithTest(void)
{
	utCyclic(&Testsuite);
}

void _EXIT exitTestSuite(void)
{
	utExit(&Testsuite);
}
```

#### autoGeneratedFile.c - Auto generated code - list of all test sets in the program
```c
/*
B+R UnitTest: This is generated code.
Do not edit! Do not move!
Description: UnitTest Testprogramm infrastructure (List of TestSets).
LastUpdated: 2022-09-26 13:08:18Z
By B+R UnitTest Helper Version: 2.0.1.59
*/
#include "UnitTest.h"

UNITTEST_TESTSET_DECLARATION  Set_AuditMgr;
UNITTEST_TESTSET_DECLARATION  Set_Common;

UNITTEST_TESTSET_FIXTURES(utTestSets)
{
	new_TestSet(Set_AuditMgr),
	new_TestSet(Set_Common),
};
UNTITTEST_TESTSET_HANDLER();
```
